LIN {X 0,Y 157.357,Z 221.695,A -85,B 0,C 180,E1 -23600.932,E2 -23600.932} C_VEL
LIN {X 0,Y 157.308,Z 221.703,A -85,B 0,C 180,E1 -23606.678,E2 -23606.678} C_VEL
LIN {X 0,Y 157.277,Z 221.702,A -85,B 0,C 180,E1 -23612.424,E2 -23612.424} C_VEL
LIN {X 0,Y 157.281,Z 221.706,A -85,B 0,C 180,E1 -23616.454,E2 -23616.454} C_VEL
LIN {X 0,Y 157.21,Z 221.714,A -85,B 0,C 180,E1 -23622.107,E2 -23622.107} C_VEL
LIN {X 0,Y 157.207,Z 221.711,A -85,B 0,C 180,E1 -23627.887,E2 -23627.887} C_VEL
LIN {X 0,Y 157.263,Z 221.709,A -85,B 0,C 180,E1 -23633.549,E2 -23633.549} C_VEL
LIN {X 0,Y 157.289,Z 221.703,A -85,B 0,C 180,E1 -23638.094,E2 -23638.094} C_VEL
LIN {X 0,Y 157.317,Z 221.699,A -85,B 0,C 180,E1 -23643.465,E2 -23643.465} C_VEL
LIN {X 0,Y 157.388,Z 221.692,A -85,B 0,C 180,E1 -23649.666,E2 -23649.666} C_VEL
LIN {X 0,Y 157.456,Z 221.679,A -85,B 0,C 180,E1 -23654.466,E2 -23654.466} C_VEL
LIN {X 0,Y 157.728,Z 221.648,A -85,B 0,C 180,E1 -23659.733,E2 -23659.733} C_VEL
LIN {X 0,Y 157.802,Z 221.635,A -85,B 0,C 180,E1 -23662.321,E2 -23662.321} C_VEL
LIN {X 0,Y 158.251,Z 221.58,A -85,B 0,C 180,E1 -23670,E2 -23670} C_VEL
LIN {X 0,Y 157.71,Z 221.652,A -85,B 0,C 180,E1 -23675.113,E2 -23675.113} C_VEL
LIN {X 0,Y 157.744,Z 221.644,A -85,B 0,C 180,E1 -23677.681,E2 -23677.681} C_VEL
LIN {X 0,Y 157.517,Z 221.675,A -85,B 0,C 180,E1 -23681.027,E2 -23681.027} C_VEL
LIN {X 0,Y 156.597,Z 221.813,A -85,B 0,C 180,E1 -23686.708,E2 -23686.708} C_VEL
LIN {X 0,Y 156.129,Z 224.06,A -85,B 0,C 180,E1 -23690.029,E2 -23690.029} C_VEL
LIN {X 0,Y 157.923,Z 235.315,A -85,B 0,C 180,E1 -23691.539,E2 -23691.539} C_VEL
LIN {X 0,Y 159.098,Z 244.23,A -85,B 0,C 180,E1 -23693.081,E2 -23693.081} C_VEL
LIN {X 0,Y 160.081,Z 253.236,A -85,B 0,C 180,E1 -23694.996,E2 -23694.996} C_VEL
LIN {X 0,Y 160.318,Z 256.028,A -85,B 0,C 180,E1 -23695.651,E2 -23695.651} C_VEL
LIN {X 0,Y 159.013,Z 264.361,A -85,B 0,C 180,E1 -23697.883,E2 -23697.883} C_VEL
LIN {X 0,Y 157.724,Z 272.061,A -85,B 0,C 180,E1 -23700.454,E2 -23700.454} C_VEL
LIN {X 0,Y 156.614,Z 279.016,A -85,B 0,C 180,E1 -23703.347,E2 -23703.347} C_VEL
LIN {X 0,Y 155.581,Z 285.499,A -85,B 0,C 180,E1 -23706.765,E2 -23706.765} C_VEL
LIN {X 0,Y 154.989,Z 289.667,A -85,B 0,C 180,E1 -23709.572,E2 -23709.572} C_VEL
LIN {X 0,Y 154.605,Z 293.901,A -85,B 0,C 180,E1 -23713.341,E2 -23713.341} C_VEL
LIN {X 0,Y 154.717,Z 296.859,A -85,B 0,C 180,E1 -23717.053,E2 -23717.053} C_VEL
LIN {X 0,Y 155.31,Z 298.71,A -85,B 0,C 180,E1 -23720.693,E2 -23720.693} C_VEL
LIN {X 0,Y 156.458,Z 299.555,A -85,B 0,C 180,E1 -23724.274,E2 -23724.274} C_VEL
LIN {X 0,Y 158.08,Z 299.423,A -85,B 0,C 180,E1 -23727.761,E2 -23727.761} C_VEL
LIN {X 0,Y 160.289,Z 298.258,A -85,B 0,C 180,E1 -23731.272,E2 -23731.272} C_VEL
LIN {X 0,Y 163.108,Z 295.89,A -85,B 0,C 180,E1 -23734.802,E2 -23734.802} C_VEL
LIN {X 0,Y 166.573,Z 292.371,A -85,B 0,C 180,E1 -23738.158,E2 -23738.158} C_VEL
LIN {X 0,Y 169.515,Z 288.835,A -85,B 0,C 180,E1 -23740.632,E2 -23740.632} C_VEL
LIN {X 0,Y 172.744,Z 284.45,A -85,B 0,C 180,E1 -23743.01,E2 -23743.01} C_VEL
LIN {X 0,Y 175.017,Z 281.08,A -85,B 0,C 180,E1 -23744.523,E2 -23744.523} C_VEL
LIN {X 0,Y 176.013,Z 277.817,A -85,B 0,C 180,E1 -23746.141,E2 -23746.141} C_VEL
LIN {X 0,Y 176.892,Z 271.671,A -85,B 0,C 180,E1 -23749.124,E2 -23749.124} C_VEL
LIN {X 0,Y 176.984,Z 265.582,A -85,B 0,C 180,E1 -23752.013,E2 -23752.013} C_VEL
LIN {X 0,Y 176.219,Z 259.844,A -85,B 0,C 180,E1 -23754.854,E2 -23754.854} C_VEL
LIN {X 0,Y 174.297,Z 253.46,A -85,B 0,C 180,E1 -23758.584,E2 -23758.584} C_VEL
LIN {X 0,Y 172.739,Z 249.567,A -85,B 0,C 180,E1 -23761.168,E2 -23761.168} C_VEL
LIN {X 0,Y 171.244,Z 246.223,A -85,B 0,C 180,E1 -23763.734,E2 -23763.734} C_VEL
LIN {X 0,Y 168.915,Z 243.311,A -85,B 0,C 180,E1 -23767.172,E2 -23767.172} C_VEL
LIN {X 0,Y 167.788,Z 240.918,A -85,B 0,C 180,E1 -23769.647,E2 -23769.647} C_VEL
LIN {X 0,Y 164.941,Z 238.279,A -85,B 0,C 180,E1 -23777.355,E2 -23777.355} C_VEL
LIN {X 0,Y 164.603,Z 237.817,A -85,B 0,C 180,E1 -23780.062,E2 -23780.062} C_VEL
LIN {X 0,Y 164.625,Z 238.233,A -85,B 0,C 180,E1 -23783.929,E2 -23783.929} C_VEL
LIN {X 0,Y 164.925,Z 239.123,A -85,B 0,C 180,E1 -23786.508,E2 -23786.508} C_VEL
LIN {X 0,Y 167.958,Z 244.088,A -85,B 0,C 180,E1 -23794.624,E2 -23794.624} C_VEL
LIN {X 0,Y 169.814,Z 248.809,A -85,B 0,C 180,E1 -23798.376,E2 -23798.376} C_VEL
LIN {X 0,Y 170.797,Z 250.242,A -85,B 0,C 180,E1 -23799.699,E2 -23799.699} C_VEL
LIN {X 0,Y 173.191,Z 256.311,A -85,B 0,C 180,E1 -23803.621,E2 -23803.621} C_VEL
LIN {X 0,Y 175.702,Z 263.842,A -85,B 0,C 180,E1 -23807.731,E2 -23807.731} C_VEL
LIN {X 0,Y 176.827,Z 268.296,A -85,B 0,C 180,E1 -23809.866,E2 -23809.866} C_VEL
LIN {X 0,Y 176.722,Z 272.386,A -85,B 0,C 180,E1 -23811.419,E2 -23811.419} C_VEL
LIN {X 0,Y 175.572,Z 280.289,A -85,B 0,C 180,E1 -23814.316,E2 -23814.316} C_VEL
LIN {X 0,Y 173.444,Z 288.286,A -85,B 0,C 180,E1 -23817.528,E2 -23817.528} C_VEL
LIN {X 0,Y 171.758,Z 292.829,A -85,B 0,C 180,E1 -23819.555,E2 -23819.555} C_VEL
LIN {X 0,Y 168.933,Z 297.944,A -85,B 0,C 180,E1 -23822.094,E2 -23822.094} C_VEL
LIN {X 0,Y 165.345,Z 302.617,A -85,B 0,C 180,E1 -23824.846,E2 -23824.846} C_VEL
LIN {X 0,Y 161.783,Z 306.868,A -85,B 0,C 180,E1 -23828.331,E2 -23828.331} C_VEL
LIN {X 0,Y 158.947,Z 309.905,A -85,B 0,C 180,E1 -23831.971,E2 -23831.971} C_VEL
LIN {X 0,Y 157.539,Z 311.3,A -85,B 0,C 180,E1 -23834.475,E2 -23834.475} C_VEL
LIN {X 0,Y 156.396,Z 312.246,A -85,B 0,C 180,E1 -23837.016,E2 -23837.016} C_VEL
LIN {X 0,Y 155.614,Z 312.675,A -85,B 0,C 180,E1 -23839.593,E2 -23839.593} C_VEL
LIN {X 0,Y 155.132,Z 312.568,A -85,B 0,C 180,E1 -23842.189,E2 -23842.189} C_VEL
LIN {X 0,Y 154.948,Z 311.55,A -85,B 0,C 180,E1 -23846.274,E2 -23846.274} C_VEL
LIN {X 0,Y 155.245,Z 309.496,A -85,B 0,C 180,E1 -23850,E2 -23850} C_VEL
LIN {X 0,Y 155.182,Z 306.489,A -85,B 0,C 180,E1 -23853.423,E2 -23853.423} C_VEL
LIN {X 0,Y 155.219,Z 302.834,A -85,B 0,C 180,E1 -23856.5,E2 -23856.5} C_VEL
LIN {X 0,Y 155.653,Z 297.85,A -85,B 0,C 180,E1 -23859.749,E2 -23859.749} C_VEL
LIN {X 0,Y 156.199,Z 292.931,A -85,B 0,C 180,E1 -23862.341,E2 -23862.341} C_VEL
LIN {X 0,Y 157.058,Z 286.99,A -85,B 0,C 180,E1 -23864.91,E2 -23864.91} C_VEL
LIN {X 0,Y 158.18,Z 279.751,A -85,B 0,C 180,E1 -23867.452,E2 -23867.452} C_VEL
LIN {X 0,Y 158.643,Z 275.533,A -85,B 0,C 180,E1 -23868.735,E2 -23868.735} C_VEL
LIN {X 0,Y 158.451,Z 266.744,A -85,B 0,C 180,E1 -23870.973,E2 -23870.973} C_VEL
LIN {X 0,Y 158.166,Z 258.965,A -85,B 0,C 180,E1 -23872.606,E2 -23872.606} C_VEL
LIN {X 0,Y 157.761,Z 249.777,A -85,B 0,C 180,E1 -23874.161,E2 -23874.161} C_VEL
LIN {X 0,Y 157.069,Z 239.045,A -85,B 0,C 180,E1 -23875.555,E2 -23875.555} C_VEL
LIN {X 0,Y 156.809,Z 235.295,A -85,B 0,C 180,E1 -23875.97,E2 -23875.97} C_VEL
LIN {X 0,Y 158.126,Z 231.22,A -85,B 0,C 180,E1 -23880.739,E2 -23880.739} C_VEL
LIN {X 0,Y 158.843,Z 228.659,A -85,B 0,C 180,E1 -23883.759,E2 -23883.759} C_VEL
LIN {X 0,Y 157.955,Z 224.322,A -85,B 0,C 180,E1 -23889.248,E2 -23889.248} C_VEL
LIN {X 0,Y 156.982,Z 223.117,A -85,B 0,C 180,E1 -23891.311,E2 -23891.311} C_VEL
LIN {X 0,Y 155.184,Z 222.534,A -85,B 0,C 180,E1 -23893.376,E2 -23893.376} C_VEL
LIN {X 0,Y 151.248,Z 222.465,A -85,B 0,C 180,E1 -23897.633,E2 -23897.633} C_VEL
LIN {X 0,Y 150.18,Z 222.59,A -85,B 0,C 180,E1 -23899.886,E2 -23899.886} C_VEL
LIN {X 0,Y 150.096,Z 222.591,A -85,B 0,C 180,E1 -23900.651,E2 -23900.651} C_VEL
LIN {X 0,Y 150.194,Z 222.584,A -85,B 0,C 180,E1 -23905.837,E2 -23905.837} C_VEL
LIN {X 0,Y 150.21,Z 222.586,A -85,B 0,C 180,E1 -23909.023,E2 -23909.023} C_VEL
LIN {X 0,Y 150.246,Z 222.576,A -85,B 0,C 180,E1 -23912.719,E2 -23912.719} C_VEL
LIN {X 0,Y 150.354,Z 222.568,A -85,B 0,C 180,E1 -23919.207,E2 -23919.207} C_VEL
LIN {X 0,Y 150.366,Z 222.566,A -85,B 0,C 180,E1 -23923.712,E2 -23923.712} C_VEL
LIN {X 0,Y 150.615,Z 222.532,A -85,B 0,C 180,E1 -23929.241,E2 -23929.241} C_VEL
LIN {X 0,Y 150.707,Z 222.523,A -85,B 0,C 180,E1 -23931.956,E2 -23931.956} C_VEL
LIN {X 0,Y 151.22,Z 222.458,A -85,B 0,C 180,E1 -23939.998,E2 -23939.998} C_VEL
LIN {X 0,Y 150.706,Z 222.521,A -85,B 0,C 180,E1 -23948.04,E2 -23948.04} C_VEL
LIN {X 0,Y 150.576,Z 222.54,A -85,B 0,C 180,E1 -23951.43,E2 -23951.43} C_VEL
LIN {X 0,Y 150.329,Z 222.568,A -85,B 0,C 180,E1 -23956.288,E2 -23956.288} C_VEL
LIN {X 0,Y 150.339,Z 222.57,A -85,B 0,C 180,E1 -23960.777,E2 -23960.777} C_VEL
LIN {X 0,Y 150.24,Z 222.582,A -85,B 0,C 180,E1 -23967.277,E2 -23967.277} C_VEL
LIN {X 0,Y 150.217,Z 222.583,A -85,B 0,C 180,E1 -23972.632,E2 -23972.632} C_VEL
LIN {X 0,Y 150.209,Z 222.586,A -85,B 0,C 180,E1 -23977.459,E2 -23977.459} C_VEL
LIN {X 0,Y 150.151,Z 222.59,A -85,B 0,C 180,E1 -23981.504,E2 -23981.504} C_VEL
LIN {X 0,Y 150.122,Z 222.597,A -85,B 0,C 180,E1 -23985.393,E2 -23985.393} C_VEL
LIN {X 0,Y 150.146,Z 222.589,A -85,B 0,C 180,E1 -23989.056,E2 -23989.056} C_VEL
LIN {X 0,Y 150.175,Z 222.59,A -85,B 0,C 180,E1 -23992.705,E2 -23992.705} C_VEL
LIN {X 0,Y 150.21,Z 222.581,A -85,B 0,C 180,E1 -23997.366,E2 -23997.366} C_VEL
LIN {X 0,Y 150.239,Z 222.581,A -85,B 0,C 180,E1 -24002.716,E2 -24002.716} C_VEL
LIN {X 0,Y 150.345,Z 222.571,A -85,B 0,C 180,E1 -24009.206,E2 -24009.206} C_VEL
LIN {X 0,Y 150.362,Z 222.563,A -85,B 0,C 180,E1 -24013.713,E2 -24013.713} C_VEL
LIN {X 0,Y 150.652,Z 222.53,A -85,B 0,C 180,E1 -24019.245,E2 -24019.245} C_VEL
LIN {X 0,Y 150.738,Z 222.514,A -85,B 0,C 180,E1 -24021.959,E2 -24021.959} C_VEL
LIN {X 0,Y 151.211,Z 222.456,A -85,B 0,C 180,E1 -24030,E2 -24030} C_VEL
LIN {X 0,Y 150.654,Z 222.527,A -85,B 0,C 180,E1 -24038.044,E2 -24038.044} C_VEL
LIN {X 0,Y 150.433,Z 222.558,A -85,B 0,C 180,E1 -24041.177,E2 -24041.177} C_VEL
LIN {X 0,Y 149.471,Z 222.712,A -85,B 0,C 180,E1 -24046.913,E2 -24046.913} C_VEL
LIN {X 0,Y 149.11,Z 224.303,A -85,B 0,C 180,E1 -24049.354,E2 -24049.354} C_VEL
LIN {X 0,Y 150.794,Z 234.895,A -85,B 0,C 180,E1 -24050.816,E2 -24050.816} C_VEL
LIN {X 0,Y 151.854,Z 242.993,A -85,B 0,C 180,E1 -24052.245,E2 -24052.245} C_VEL
LIN {X 0,Y 152.818,Z 251.392,A -85,B 0,C 180,E1 -24054.053,E2 -24054.053} C_VEL
LIN {X 0,Y 153.211,Z 257.128,A -85,B 0,C 180,E1 -24055.47,E2 -24055.47} C_VEL
LIN {X 0,Y 151.953,Z 264.547,A -85,B 0,C 180,E1 -24057.549,E2 -24057.549} C_VEL
LIN {X 0,Y 150.658,Z 272.211,A -85,B 0,C 180,E1 -24060.216,E2 -24060.216} C_VEL
LIN {X 0,Y 149.479,Z 279.357,A -85,B 0,C 180,E1 -24063.322,E2 -24063.322} C_VEL
LIN {X 0,Y 148.373,Z 286.201,A -85,B 0,C 180,E1 -24067.166,E2 -24067.166} C_VEL
LIN {X 0,Y 147.739,Z 290.657,A -85,B 0,C 180,E1 -24070.441,E2 -24070.441} C_VEL
LIN {X 0,Y 147.492,Z 294.709,A -85,B 0,C 180,E1 -24074.381,E2 -24074.381} C_VEL
LIN {X 0,Y 147.734,Z 297.522,A -85,B 0,C 180,E1 -24078.244,E2 -24078.244} C_VEL
LIN {X 0,Y 148.531,Z 299.257,A -85,B 0,C 180,E1 -24082.043,E2 -24082.043} C_VEL
LIN {X 0,Y 149.895,Z 299.978,A -85,B 0,C 180,E1 -24085.765,E2 -24085.765} C_VEL
LIN {X 0,Y 151.779,Z 299.699,A -85,B 0,C 180,E1 -24089.383,E2 -24089.383} C_VEL
LIN {X 0,Y 154.19,Z 298.452,A -85,B 0,C 180,E1 -24092.886,E2 -24092.886} C_VEL
LIN {X 0,Y 157.064,Z 296.25,A -85,B 0,C 180,E1 -24096.255,E2 -24096.255} C_VEL
LIN {X 0,Y 160.567,Z 292.975,A -85,B 0,C 180,E1 -24099.505,E2 -24099.505} C_VEL
LIN {X 0,Y 164.43,Z 288.619,A -85,B 0,C 180,E1 -24102.593,E2 -24102.593} C_VEL
LIN {X 0,Y 168.84,Z 282.94,A -85,B 0,C 180,E1 -24105.539,E2 -24105.539} C_VEL
LIN {X 0,Y 170.062,Z 279.332,A -85,B 0,C 180,E1 -24107.472,E2 -24107.472} C_VEL
LIN {X 0,Y 171.082,Z 273.883,A -85,B 0,C 180,E1 -24110.37,E2 -24110.37} C_VEL
LIN {X 0,Y 171.363,Z 268.962,A -85,B 0,C 180,E1 -24112.935,E2 -24112.935} C_VEL
LIN {X 0,Y 171.142,Z 264.718,A -85,B 0,C 180,E1 -24115.291,E2 -24115.291} C_VEL
LIN {X 0,Y 169.882,Z 259.168,A -85,B 0,C 180,E1 -24118.817,E2 -24118.817} C_VEL
LIN {X 0,Y 168.254,Z 254.292,A -85,B 0,C 180,E1 -24122.396,E2 -24122.396} C_VEL
LIN {X 0,Y 167.637,Z 252.581,A -85,B 0,C 180,E1 -24123.814,E2 -24123.814} C_VEL
LIN {X 0,Y 164.769,Z 247.382,A -85,B 0,C 180,E1 -24129.826,E2 -24129.826} C_VEL
LIN {X 0,Y 162.267,Z 244.828,A -85,B 0,C 180,E1 -24137.665,E2 -24137.665} C_VEL
LIN {X 0,Y 162.024,Z 244.453,A -85,B 0,C 180,E1 -24140.307,E2 -24140.307} C_VEL
LIN {X 0,Y 162.115,Z 245.007,A -85,B 0,C 180,E1 -24144.441,E2 -24144.441} C_VEL
LIN {X 0,Y 162.645,Z 246.843,A -85,B 0,C 180,E1 -24148.382,E2 -24148.382} C_VEL
LIN {X 0,Y 164.582,Z 250.059,A -85,B 0,C 180,E1 -24153.722,E2 -24153.722} C_VEL
LIN {X 0,Y 166.942,Z 256.043,A -85,B 0,C 180,E1 -24159.161,E2 -24159.161} C_VEL
LIN {X 0,Y 168.757,Z 261.525,A -85,B 0,C 180,E1 -24162.984,E2 -24162.984} C_VEL
LIN {X 0,Y 170.316,Z 267.016,A -85,B 0,C 180,E1 -24166.231,E2 -24166.231} C_VEL
LIN {X 0,Y 171.4,Z 272.056,A -85,B 0,C 180,E1 -24169.001,E2 -24169.001} C_VEL
LIN {X 0,Y 171.045,Z 275.831,A -85,B 0,C 180,E1 -24170.555,E2 -24170.555} C_VEL
LIN {X 0,Y 169.552,Z 282.828,A -85,B 0,C 180,E1 -24173.393,E2 -24173.393} C_VEL
LIN {X 0,Y 167.996,Z 287.976,A -85,B 0,C 180,E1 -24175.615,E2 -24175.615} C_VEL
LIN {X 0,Y 165.588,Z 293.793,A -85,B 0,C 180,E1 -24178.393,E2 -24178.393} C_VEL
LIN {X 0,Y 163.418,Z 297.577,A -85,B 0,C 180,E1 -24180.359,E2 -24180.359} C_VEL
LIN {X 0,Y 158.967,Z 302.982,A -85,B 0,C 180,E1 -24183.762,E2 -24183.762} C_VEL
LIN {X 0,Y 155.217,Z 307.043,A -85,B 0,C 180,E1 -24187.365,E2 -24187.365} C_VEL
LIN {X 0,Y 152.191,Z 309.927,A -85,B 0,C 180,E1 -24191.141,E2 -24191.141} C_VEL
LIN {X 0,Y 150.691,Z 311.177,A -85,B 0,C 180,E1 -24193.75,E2 -24193.75} C_VEL
LIN {X 0,Y 149.48,Z 311.981,A -85,B 0,C 180,E1 -24196.404,E2 -24196.404} C_VEL
LIN {X 0,Y 148.616,Z 312.347,A -85,B 0,C 180,E1 -24199.097,E2 -24199.097} C_VEL
LIN {X 0,Y 148.085,Z 312.163,A -85,B 0,C 180,E1 -24201.815,E2 -24201.815} C_VEL
LIN {X 0,Y 147.889,Z 310.828,A -85,B 0,C 180,E1 -24206.368,E2 -24206.368} C_VEL
LIN {X 0,Y 148.186,Z 308.713,A -85,B 0,C 180,E1 -24210.001,E2 -24210.001} C_VEL
LIN {X 0,Y 148.14,Z 305.73,A -85,B 0,C 180,E1 -24213.412,E2 -24213.412} C_VEL
LIN {X 0,Y 148.183,Z 301.724,A -85,B 0,C 180,E1 -24216.81,E2 -24216.81} C_VEL
LIN {X 0,Y 148.656,Z 296.56,A -85,B 0,C 180,E1 -24220.212,E2 -24220.212} C_VEL
LIN {X 0,Y 149.262,Z 291.444,A -85,B 0,C 180,E1 -24222.924,E2 -24222.924} C_VEL
LIN {X 0,Y 150.193,Z 285.274,A -85,B 0,C 180,E1 -24225.609,E2 -24225.609} C_VEL
LIN {X 0,Y 151.502,Z 276.74,A -85,B 0,C 180,E1 -24228.598,E2 -24228.598} C_VEL
LIN {X 0,Y 151.432,Z 267.772,A -85,B 0,C 180,E1 -24231.081,E2 -24231.081} C_VEL
LIN {X 0,Y 151.15,Z 259.634,A -85,B 0,C 180,E1 -24232.918,E2 -24232.918} C_VEL
LIN {X 0,Y 150.775,Z 250.215,A -85,B 0,C 180,E1 -24234.621,E2 -24234.621} C_VEL
LIN {X 0,Y 150.204,Z 240.494,A -85,B 0,C 180,E1 -24235.984,E2 -24235.984} C_VEL
LIN {X 0,Y 149.858,Z 235.041,A -85,B 0,C 180,E1 -24236.662,E2 -24236.662} C_VEL
LIN {X 0,Y 151.413,Z 230.571,A -85,B 0,C 180,E1 -24242.123,E2 -24242.123} C_VEL
LIN {X 0,Y 151.753,Z 229.253,A -85,B 0,C 180,E1 -24243.763,E2 -24243.763} C_VEL
LIN {X 0,Y 151.135,Z 226.209,A -85,B 0,C 180,E1 -24247.763,E2 -24247.763} C_VEL
LIN {X 0,Y 150.464,Z 222.555,A -85,B 0,C 180,E1 -24252.807,E2 -24252.807} C_VEL
LIN {X 0,Y 150.154,Z 222.592,A -85,B 0,C 180,E1 -24259.057,E2 -24259.057} C_VEL
LIN {X 0,Y 150.096,Z 222.591,A -85,B 0,C 180,E1 -24260.651,E2 -24260.651} C_VEL
LIN {X 0,Y 149.455,Z 222.68,A -85,B 0,C 180,E1 -24262.891,E2 -24262.891} C_VEL
LIN {X 0,Y 147.93,Z 222.869,A -85,B 0,C 180,E1 -24265.102,E2 -24265.102} C_VEL
LIN {X 0,Y 143.499,Z 223.421,A -85,B 0,C 180,E1 -24271.171,E2 -24271.171} C_VEL
LIN {X 0,Y 143.163,Z 223.458,A -85,B 0,C 180,E1 -24272.77,E2 -24272.77} C_VEL
LIN {X 0,Y 143.28,Z 223.448,A -85,B 0,C 180,E1 -24278.746,E2 -24278.746} C_VEL
LIN {X 0,Y 143.305,Z 223.442,A -85,B 0,C 180,E1 -24282.885,E2 -24282.885} C_VEL
LIN {X 0,Y 143.541,Z 223.414,A -85,B 0,C 180,E1 -24288.703,E2 -24288.703} C_VEL
LIN {X 0,Y 143.629,Z 223.404,A -85,B 0,C 180,E1 -24291.556,E2 -24291.556} C_VEL
LIN {X 0,Y 144.178,Z 223.335,A -85,B 0,C 180,E1 -24299.998,E2 -24299.998} C_VEL
LIN {X 0,Y 143.627,Z 223.403,A -85,B 0,C 180,E1 -24308.439,E2 -24308.439} C_VEL
LIN {X 0,Y 143.502,Z 223.421,A -85,B 0,C 180,E1 -24311.618,E2 -24311.618} C_VEL
LIN {X 0,Y 143.268,Z 223.451,A -85,B 0,C 180,E1 -24317.115,E2 -24317.115} C_VEL
LIN {X 0,Y 143.267,Z 223.449,A -85,B 0,C 180,E1 -24321.242,E2 -24321.242} C_VEL
LIN {X 0,Y 143.187,Z 223.461,A -85,B 0,C 180,E1 -24327.933,E2 -24327.933} C_VEL
LIN {X 0,Y 143.167,Z 223.461,A -85,B 0,C 180,E1 -24333.433,E2 -24333.433} C_VEL
LIN {X 0,Y 143.072,Z 223.471,A -85,B 0,C 180,E1 -24339.683,E2 -24339.683} C_VEL
LIN {X 0,Y 143.054,Z 223.477,A -85,B 0,C 180,E1 -24343.452,E2 -24343.452} C_VEL
LIN {X 0,Y 143.061,Z 223.474,A -85,B 0,C 180,E1 -24347.463,E2 -24347.463} C_VEL
LIN {X 0,Y 143.073,Z 223.476,A -85,B 0,C 180,E1 -24351.804,E2 -24351.804} C_VEL
LIN {X 0,Y 143.177,Z 223.457,A -85,B 0,C 180,E1 -24357.319,E2 -24357.319} C_VEL
LIN {X 0,Y 143.186,Z 223.46,A -85,B 0,C 180,E1 -24362.061,E2 -24362.061} C_VEL
LIN {X 0,Y 143.271,Z 223.45,A -85,B 0,C 180,E1 -24368.744,E2 -24368.744} C_VEL
LIN {X 0,Y 143.299,Z 223.443,A -85,B 0,C 180,E1 -24372.886,E2 -24372.886} C_VEL
LIN {X 0,Y 143.588,Z 223.412,A -85,B 0,C 180,E1 -24378.709,E2 -24378.709} C_VEL
LIN {X 0,Y 143.659,Z 223.396,A -85,B 0,C 180,E1 -24381.56,E2 -24381.56} C_VEL
LIN {X 0,Y 144.17,Z 223.333,A -85,B 0,C 180,E1 -24389.999,E2 -24389.999} C_VEL
LIN {X 0,Y 143.565,Z 223.409,A -85,B 0,C 180,E1 -24398.445,E2 -24398.445} C_VEL
LIN {X 0,Y 143.336,Z 223.441,A -85,B 0,C 180,E1 -24401.31,E2 -24401.31} C_VEL
LIN {X 0,Y 142.382,Z 223.56,A -85,B 0,C 180,E1 -24407.042,E2 -24407.042} C_VEL
LIN {X 0,Y 142.126,Z 224.534,A -85,B 0,C 180,E1 -24408.628,E2 -24408.628} C_VEL
LIN {X 0,Y 143.95,Z 236.408,A -85,B 0,C 180,E1 -24410.421,E2 -24410.421} C_VEL
LIN {X 0,Y 145.022,Z 244.991,A -85,B 0,C 180,E1 -24412.06,E2 -24412.06} C_VEL
LIN {X 0,Y 145.95,Z 253.361,A -85,B 0,C 180,E1 -24414.01,E2 -24414.01} C_VEL
LIN {X 0,Y 146.104,Z 257.993,A -85,B 0,C 180,E1 -24415.233,E2 -24415.233} C_VEL
LIN {X 0,Y 144.766,Z 265.459,A -85,B 0,C 180,E1 -24417.464,E2 -24417.464} C_VEL
LIN {X 0,Y 143.528,Z 272.666,A -85,B 0,C 180,E1 -24420.125,E2 -24420.125} C_VEL
LIN {X 0,Y 142.175,Z 280.577,A -85,B 0,C 180,E1 -24423.785,E2 -24423.785} C_VEL
LIN {X 0,Y 141.092,Z 287.245,A -85,B 0,C 180,E1 -24427.903,E2 -24427.903} C_VEL
LIN {X 0,Y 140.525,Z 291.614,A -85,B 0,C 180,E1 -24431.398,E2 -24431.398} C_VEL
LIN {X 0,Y 140.414,Z 295.51,A -85,B 0,C 180,E1 -24435.519,E2 -24435.519} C_VEL
LIN {X 0,Y 140.823,Z 298.186,A -85,B 0,C 180,E1 -24439.554,E2 -24439.554} C_VEL
LIN {X 0,Y 141.844,Z 299.78,A -85,B 0,C 180,E1 -24443.521,E2 -24443.521} C_VEL
LIN {X 0,Y 143.445,Z 300.35,A -85,B 0,C 180,E1 -24447.392,E2 -24447.392} C_VEL
LIN {X 0,Y 145.616,Z 299.941,A -85,B 0,C 180,E1 -24451.145,E2 -24451.145} C_VEL
LIN {X 0,Y 148.329,Z 298.586,A -85,B 0,C 180,E1 -24454.762,E2 -24454.762} C_VEL
LIN {X 0,Y 151.549,Z 296.269,A -85,B 0,C 180,E1 -24458.226,E2 -24458.226} C_VEL
LIN {X 0,Y 155.317,Z 292.905,A -85,B 0,C 180,E1 -24461.536,E2 -24461.536} C_VEL
LIN {X 0,Y 160.083,Z 287.925,A -85,B 0,C 180,E1 -24464.982,E2 -24464.982} C_VEL
LIN {X 0,Y 163.095,Z 284.085,A -85,B 0,C 180,E1 -24466.988,E2 -24466.988} C_VEL
LIN {X 0,Y 164.871,Z 278.73,A -85,B 0,C 180,E1 -24470.185,E2 -24470.185} C_VEL
LIN {X 0,Y 165.739,Z 273.335,A -85,B 0,C 180,E1 -24473.306,E2 -24473.306} C_VEL
LIN {X 0,Y 165.75,Z 268.349,A -85,B 0,C 180,E1 -24476.356,E2 -24476.356} C_VEL
LIN {X 0,Y 164.829,Z 263.239,A -85,B 0,C 180,E1 -24480.002,E2 -24480.002} C_VEL
LIN {X 0,Y 163.638,Z 258.825,A -85,B 0,C 180,E1 -24483.696,E2 -24483.696} C_VEL
LIN {X 0,Y 162.566,Z 256.708,A -85,B 0,C 180,E1 -24486.109,E2 -24486.109} C_VEL
LIN {X 0,Y 161.318,Z 253.617,A -85,B 0,C 180,E1 -24490.038,E2 -24490.038} C_VEL
LIN {X 0,Y 159.191,Z 251.178,A -85,B 0,C 180,E1 -24498.003,E2 -24498.003} C_VEL
LIN {X 0,Y 159.005,Z 251.007,A -85,B 0,C 180,E1 -24501.846,E2 -24501.846} C_VEL
LIN {X 0,Y 159.075,Z 251.221,A -85,B 0,C 180,E1 -24503.432,E2 -24503.432} C_VEL
LIN {X 0,Y 159.204,Z 252.152,A -85,B 0,C 180,E1 -24506.198,E2 -24506.198} C_VEL
LIN {X 0,Y 160.382,Z 255.147,A -85,B 0,C 180,E1 -24511.727,E2 -24511.727} C_VEL
LIN {X 0,Y 161.35,Z 257.328,A -85,B 0,C 180,E1 -24514.491,E2 -24514.491} C_VEL
LIN {X 0,Y 162.876,Z 262.191,A -85,B 0,C 180,E1 -24519.042,E2 -24519.042} C_VEL
LIN {X 0,Y 164.073,Z 266.36,A -85,B 0,C 180,E1 -24522.182,E2 -24522.182} C_VEL
LIN {X 0,Y 165.431,Z 272.608,A -85,B 0,C 180,E1 -24526.24,E2 -24526.24} C_VEL
LIN {X 0,Y 165.855,Z 275.249,A -85,B 0,C 180,E1 -24527.879,E2 -24527.879} C_VEL
LIN {X 0,Y 165.269,Z 279.337,A -85,B 0,C 180,E1 -24529.733,E2 -24529.733} C_VEL
LIN {X 0,Y 163.201,Z 286.494,A -85,B 0,C 180,E1 -24532.923,E2 -24532.923} C_VEL
LIN {X 0,Y 160.103,Z 293.616,A -85,B 0,C 180,E1 -24536.519,E2 -24536.519} C_VEL
LIN {X 0,Y 157.306,Z 298.17,A -85,B 0,C 180,E1 -24539.084,E2 -24539.084} C_VEL
LIN {X 0,Y 152.654,Z 303.37,A -85,B 0,C 180,E1 -24542.588,E2 -24542.588} C_VEL
LIN {X 0,Y 148.701,Z 307.261,A -85,B 0,C 180,E1 -24546.314,E2 -24546.314} C_VEL
LIN {X 0,Y 145.473,Z 309.961,A -85,B 0,C 180,E1 -24550.234,E2 -24550.234} C_VEL
LIN {X 0,Y 143.876,Z 311.06,A -85,B 0,C 180,E1 -24552.958,E2 -24552.958} C_VEL
LIN {X 0,Y 142.589,Z 311.717,A -85,B 0,C 180,E1 -24555.733,E2 -24555.733} C_VEL
LIN {X 0,Y 141.642,Z 311.944,A -85,B 0,C 180,E1 -24558.553,E2 -24558.553} C_VEL
LIN {X 0,Y 141.048,Z 311.72,A -85,B 0,C 180,E1 -24561.404,E2 -24561.404} C_VEL
LIN {X 0,Y 140.85,Z 310.051,A -85,B 0,C 180,E1 -24566.351,E2 -24566.351} C_VEL
LIN {X 0,Y 141.127,Z 307.88,A -85,B 0,C 180,E1 -24570.001,E2 -24570.001} C_VEL
LIN {X 0,Y 141.121,Z 305.505,A -85,B 0,C 180,E1 -24572.855,E2 -24572.855} C_VEL
LIN {X 0,Y 141.054,Z 302.461,A -85,B 0,C 180,E1 -24575.72,E2 -24575.72} C_VEL
LIN {X 0,Y 141.426,Z 297.571,A -85,B 0,C 180,E1 -24579.295,E2 -24579.295} C_VEL
LIN {X 0,Y 141.979,Z 292.756,A -85,B 0,C 180,E1 -24582.145,E2 -24582.145} C_VEL
LIN {X 0,Y 142.812,Z 286.904,A -85,B 0,C 180,E1 -24584.973,E2 -24584.973} C_VEL
LIN {X 0,Y 143.987,Z 279.782,A -85,B 0,C 180,E1 -24587.762,E2 -24587.762} C_VEL
LIN {X 0,Y 144.464,Z 275.668,A -85,B 0,C 180,E1 -24589.171,E2 -24589.171} C_VEL
LIN {X 0,Y 144.326,Z 266.004,A -85,B 0,C 180,E1 -24591.89,E2 -24591.89} C_VEL
LIN {X 0,Y 144.066,Z 257.989,A -85,B 0,C 180,E1 -24593.733,E2 -24593.733} C_VEL
LIN {X 0,Y 143.745,Z 249.405,A -85,B 0,C 180,E1 -24595.329,E2 -24595.329} C_VEL
LIN {X 0,Y 143.193,Z 239.472,A -85,B 0,C 180,E1 -24596.762,E2 -24596.762} C_VEL
LIN {X 0,Y 142.909,Z 234.747,A -85,B 0,C 180,E1 -24597.394,E2 -24597.394} C_VEL
LIN {X 0,Y 144.357,Z 230.89,A -85,B 0,C 180,E1 -24602.381,E2 -24602.381} C_VEL
LIN {X 0,Y 144.6,Z 229.445,A -85,B 0,C 180,E1 -24604.281,E2 -24604.281} C_VEL
LIN {X 0,Y 143.819,Z 225.744,A -85,B 0,C 180,E1 -24609.441,E2 -24609.441} C_VEL
LIN {X 0,Y 143.427,Z 223.431,A -85,B 0,C 180,E1 -24612.884,E2 -24612.884} C_VEL
LIN {X 0,Y 143.065,Z 223.478,A -85,B 0,C 180,E1 -24620.308,E2 -24620.308} C_VEL
LIN {X 0,Y 143.168,Z 223.462,A -85,B 0,C 180,E1 -24626.566,E2 -24626.566} C_VEL
LIN {X 0,Y 143.163,Z 223.458,A -85,B 0,C 180,E1 -24632.77,E2 -24632.77} C_VEL
LIN {X 0,Y 142.472,Z 223.549,A -85,B 0,C 180,E1 -24635.118,E2 -24635.118} C_VEL
LIN {X 0,Y 140.921,Z 223.747,A -85,B 0,C 180,E1 -24637.437,E2 -24637.437} C_VEL
LIN {X 0,Y 136.556,Z 224.292,A -85,B 0,C 180,E1 -24643.817,E2 -24643.817} C_VEL
LIN {X 0,Y 136.273,Z 224.319,A -85,B 0,C 180,E1 -24645.497,E2 -24645.497} C_VEL
LIN {X 0,Y 136.449,Z 224.298,A -85,B 0,C 180,E1 -24648.136,E2 -24648.136} C_VEL
LIN {X 0,Y 136.555,Z 224.283,A -85,B 0,C 180,E1 -24651.116,E2 -24651.116} C_VEL
LIN {X 0,Y 137.135,Z 224.213,A -85,B 0,C 180,E1 -24659.997,E2 -24659.997} C_VEL
LIN {X 0,Y 136.552,Z 224.286,A -85,B 0,C 180,E1 -24668.88,E2 -24668.88} C_VEL
LIN {X 0,Y 136.417,Z 224.304,A -85,B 0,C 180,E1 -24671.89,E2 -24671.89} C_VEL
LIN {X 0,Y 136.188,Z 224.332,A -85,B 0,C 180,E1 -24678.034,E2 -24678.034} C_VEL
LIN {X 0,Y 136.189,Z 224.33,A -85,B 0,C 180,E1 -24681.737,E2 -24681.737} C_VEL
LIN {X 0,Y 136.113,Z 224.342,A -85,B 0,C 180,E1 -24688.624,E2 -24688.624} C_VEL
LIN {X 0,Y 136.077,Z 224.347,A -85,B 0,C 180,E1 -24694.616,E2 -24694.616} C_VEL
LIN {X 0,Y 136.048,Z 224.346,A -85,B 0,C 180,E1 -24699.205,E2 -24699.205} C_VEL
LIN {X 0,Y 135.995,Z 224.357,A -85,B 0,C 180,E1 -24703.655,E2 -24703.655} C_VEL
LIN {X 0,Y 136.001,Z 224.352,A -85,B 0,C 180,E1 -24707.794,E2 -24707.794} C_VEL
LIN {X 0,Y 136.023,Z 224.354,A -85,B 0,C 180,E1 -24711.682,E2 -24711.682} C_VEL
LIN {X 0,Y 136.051,Z 224.346,A -85,B 0,C 180,E1 -24715.737,E2 -24715.737} C_VEL
LIN {X 0,Y 136.142,Z 224.338,A -85,B 0,C 180,E1 -24722.315,E2 -24722.315} C_VEL
LIN {X 0,Y 136.238,Z 224.327,A -85,B 0,C 180,E1 -24728.831,E2 -24728.831} C_VEL
LIN {X 0,Y 136.27,Z 224.32,A -85,B 0,C 180,E1 -24735.056,E2 -24735.056} C_VEL
LIN {X 0,Y 136.491,Z 224.295,A -85,B 0,C 180,E1 -24738.114,E2 -24738.114} C_VEL
LIN {X 0,Y 136.586,Z 224.278,A -85,B 0,C 180,E1 -24741.119,E2 -24741.119} C_VEL
LIN {X 0,Y 137.127,Z 224.21,A -85,B 0,C 180,E1 -24749.999,E2 -24749.999} C_VEL
LIN {X 0,Y 136.528,Z 224.29,A -85,B 0,C 180,E1 -24755.909,E2 -24755.909} C_VEL
LIN {X 0,Y 136.466,Z 224.294,A -85,B 0,C 180,E1 -24758.887,E2 -24758.887} C_VEL
LIN {X 0,Y 136.15,Z 224.337,A -85,B 0,C 180,E1 -24761.915,E2 -24761.915} C_VEL
LIN {X 0,Y 135.311,Z 224.44,A -85,B 0,C 180,E1 -24766.987,E2 -24766.987} C_VEL
LIN {X 0,Y 135.148,Z 224.803,A -85,B 0,C 180,E1 -24767.886,E2 -24767.886} C_VEL
LIN {X 0,Y 136.773,Z 235.484,A -85,B 0,C 180,E1 -24769.532,E2 -24769.532} C_VEL
LIN {X 0,Y 137.936,Z 244.668,A -85,B 0,C 180,E1 -24771.354,E2 -24771.354} C_VEL
LIN {X 0,Y 138.903,Z 253.821,A -85,B 0,C 180,E1 -24773.588,E2 -24773.588} C_VEL
LIN {X 0,Y 139.149,Z 257.583,A -85,B 0,C 180,E1 -24774.622,E2 -24774.622} C_VEL
LIN {X 0,Y 137.581,Z 266.308,A -85,B 0,C 180,E1 -24777.37,E2 -24777.37} C_VEL
LIN {X 0,Y 136.429,Z 272.812,A -85,B 0,C 180,E1 -24779.902,E2 -24779.902} C_VEL
LIN {X 0,Y 135.295,Z 279.364,A -85,B 0,C 180,E1 -24783.027,E2 -24783.027} C_VEL
LIN {X 0,Y 134.283,Z 285.314,A -85,B 0,C 180,E1 -24786.551,E2 -24786.551} C_VEL
LIN {X 0,Y 133.519,Z 290.842,A -85,B 0,C 180,E1 -24790.779,E2 -24790.779} C_VEL
LIN {X 0,Y 133.316,Z 294.892,A -85,B 0,C 180,E1 -24795.007,E2 -24795.007} C_VEL
LIN {X 0,Y 133.454,Z 296.815,A -85,B 0,C 180,E1 -24797.499,E2 -24797.499} C_VEL
LIN {X 0,Y 134.197,Z 299.112,A -85,B 0,C 180,E1 -24801.772,E2 -24801.772} C_VEL
LIN {X 0,Y 135.613,Z 300.37,A -85,B 0,C 180,E1 -24806.014,E2 -24806.014} C_VEL
LIN {X 0,Y 137.7,Z 300.612,A -85,B 0,C 180,E1 -24810.187,E2 -24810.187} C_VEL
LIN {X 0,Y 140.487,Z 299.825,A -85,B 0,C 180,E1 -24814.218,E2 -24814.218} C_VEL
LIN {X 0,Y 143.884,Z 297.993,A -85,B 0,C 180,E1 -24818.132,E2 -24818.132} C_VEL
LIN {X 0,Y 147.953,Z 295.048,A -85,B 0,C 180,E1 -24821.81,E2 -24821.81} C_VEL
LIN {X 0,Y 152.579,Z 290.754,A -85,B 0,C 180,E1 -24825.304,E2 -24825.304} C_VEL
LIN {X 0,Y 156.27,Z 286.849,A -85,B 0,C 180,E1 -24827.663,E2 -24827.663} C_VEL
LIN {X 0,Y 157.56,Z 284.793,A -85,B 0,C 180,E1 -24828.906,E2 -24828.906} C_VEL
LIN {X 0,Y 158.849,Z 281.437,A -85,B 0,C 180,E1 -24831.094,E2 -24831.094} C_VEL
LIN {X 0,Y 159.875,Z 277.488,A -85,B 0,C 180,E1 -24833.693,E2 -24833.693} C_VEL
LIN {X 0,Y 160.31,Z 273.673,A -85,B 0,C 180,E1 -24836.232,E2 -24836.232} C_VEL
LIN {X 0,Y 159.957,Z 268.758,A -85,B 0,C 180,E1 -24840.002,E2 -24840.002} C_VEL
LIN {X 0,Y 159.172,Z 264.479,A -85,B 0,C 180,E1 -24843.8,E2 -24843.8} C_VEL
LIN {X 0,Y 158.851,Z 263.296,A -85,B 0,C 180,E1 -24845.079,E2 -24845.079} C_VEL
LIN {X 0,Y 157.309,Z 259.407,A -85,B 0,C 180,E1 -24850.619,E2 -24850.619} C_VEL
LIN {X 0,Y 155.691,Z 257.331,A -85,B 0,C 180,E1 -24858.568,E2 -24858.568} C_VEL
LIN {X 0,Y 155.606,Z 257.195,A -85,B 0,C 180,E1 -24861.184,E2 -24861.184} C_VEL
LIN {X 0,Y 155.69,Z 258.147,A -85,B 0,C 180,E1 -24865.47,E2 -24865.47} C_VEL
LIN {X 0,Y 156.863,Z 261.83,A -85,B 0,C 180,E1 -24872.526,E2 -24872.526} C_VEL
LIN {X 0,Y 157.288,Z 262.974,A -85,B 0,C 180,E1 -24873.996,E2 -24873.996} C_VEL
LIN {X 0,Y 158.465,Z 268.232,A -85,B 0,C 180,E1 -24879.109,E2 -24879.109} C_VEL
LIN {X 0,Y 159.16,Z 271.107,A -85,B 0,C 180,E1 -24881.482,E2 -24881.482} C_VEL
LIN {X 0,Y 159.957,Z 276.4,A -85,B 0,C 180,E1 -24885.333,E2 -24885.333} C_VEL
LIN {X 0,Y 160.21,Z 279.749,A -85,B 0,C 180,E1 -24887.457,E2 -24887.457} C_VEL
LIN {X 0,Y 158.355,Z 285.665,A -85,B 0,C 180,E1 -24890.341,E2 -24890.341} C_VEL
LIN {X 0,Y 155.272,Z 292.608,A -85,B 0,C 180,E1 -24893.956,E2 -24893.956} C_VEL
LIN {X 0,Y 152.71,Z 296.946,A -85,B 0,C 180,E1 -24896.478,E2 -24896.478} C_VEL
LIN {X 0,Y 149.653,Z 300.668,A -85,B 0,C 180,E1 -24898.897,E2 -24898.897} C_VEL
LIN {X 0,Y 144.97,Z 305.146,A -85,B 0,C 180,E1 -24902.578,E2 -24902.578} C_VEL
LIN {X 0,Y 140.99,Z 308.35,A -85,B 0,C 180,E1 -24906.499,E2 -24906.499} C_VEL
LIN {X 0,Y 138.795,Z 309.909,A -85,B 0,C 180,E1 -24909.241,E2 -24909.241} C_VEL
LIN {X 0,Y 137.075,Z 310.955,A -85,B 0,C 180,E1 -24912.084,E2 -24912.084} C_VEL
LIN {X 0,Y 135.708,Z 311.459,A -85,B 0,C 180,E1 -24914.993,E2 -24914.993} C_VEL
LIN {X 0,Y 134.694,Z 311.534,A -85,B 0,C 180,E1 -24917.954,E2 -24917.954} C_VEL
LIN {X 0,Y 134.035,Z 311.184,A -85,B 0,C 180,E1 -24920.95,E2 -24920.95} C_VEL
LIN {X 0,Y 133.768,Z 310.364,A -85,B 0,C 180,E1 -24923.969,E2 -24923.969} C_VEL
LIN {X 0,Y 133.855,Z 308.963,A -85,B 0,C 180,E1 -24926.991,E2 -24926.991} C_VEL
LIN {X 0,Y 134.064,Z 305.923,A -85,B 0,C 180,E1 -24931.503,E2 -24931.503} C_VEL
LIN {X 0,Y 134.007,Z 301.274,A -85,B 0,C 180,E1 -24936.021,E2 -24936.021} C_VEL
LIN {X 0,Y 134.449,Z 296.192,A -85,B 0,C 180,E1 -24939.782,E2 -24939.782} C_VEL
LIN {X 0,Y 135.062,Z 291.162,A -85,B 0,C 180,E1 -24942.777,E2 -24942.777} C_VEL
LIN {X 0,Y 135.969,Z 285.078,A -85,B 0,C 180,E1 -24945.746,E2 -24945.746} C_VEL
LIN {X 0,Y 137.252,Z 277.692,A -85,B 0,C 180,E1 -24948.665,E2 -24948.665} C_VEL
LIN {X 0,Y 137.332,Z 268.879,A -85,B 0,C 180,E1 -24951.508,E2 -24951.508} C_VEL
LIN {X 0,Y 137.07,Z 259.031,A -85,B 0,C 180,E1 -24953.998,E2 -24953.998} C_VEL
LIN {X 0,Y 136.754,Z 249.445,A -85,B 0,C 180,E1 -24955.902,E2 -24955.902} C_VEL
LIN {X 0,Y 136.213,Z 239.267,A -85,B 0,C 180,E1 -24957.461,E2 -24957.461} C_VEL
LIN {X 0,Y 135.968,Z 234.587,A -85,B 0,C 180,E1 -24958.043,E2 -24958.043} C_VEL
LIN {X 0,Y 137.264,Z 231.279,A -85,B 0,C 180,E1 -24962.522,E2 -24962.522} C_VEL
LIN {X 0,Y 137.418,Z 229.453,A -85,B 0,C 180,E1 -24965.082,E2 -24965.082} C_VEL
LIN {X 0,Y 136.752,Z 226.409,A -85,B 0,C 180,E1 -24969.564,E2 -24969.564} C_VEL
LIN {X 0,Y 136.39,Z 224.308,A -85,B 0,C 180,E1 -24972.915,E2 -24972.915} C_VEL
LIN {X 0,Y 136.068,Z 224.344,A -85,B 0,C 180,E1 -24977.817,E2 -24977.817} C_VEL
LIN {X 0,Y 136.031,Z 224.353,A -85,B 0,C 180,E1 -24981.683,E2 -24981.683} C_VEL
LIN {X 0,Y 136.089,Z 224.34,A -85,B 0,C 180,E1 -24985.72,E2 -24985.72} C_VEL
LIN {X 0,Y 136.149,Z 224.333,A -85,B 0,C 180,E1 -24992.314,E2 -24992.314} C_VEL
LIN {X 0,Y 136.246,Z 224.325,A -85,B 0,C 180,E1 -24998.831,E2 -24998.831} C_VEL
LIN {X 0,Y 136.272,Z 224.322,A -85,B 0,C 180,E1 -25005.054,E2 -25005.054} C_VEL
LIN {X 0,Y 136.273,Z 224.319,A -85,B 0,C 180,E1 -25005.497,E2 -25005.497} C_VEL
LIN {X 0,Y 135.631,Z 224.401,A -85,B 0,C 180,E1 -25007.967,E2 -25007.967} C_VEL
LIN {X 0,Y 134.09,Z 224.593,A -85,B 0,C 180,E1 -25010.406,E2 -25010.406} C_VEL
LIN {X 0,Y 130.617,Z 225.027,A -85,B 0,C 180,E1 -25015.399,E2 -25015.399} C_VEL
LIN {X 0,Y 129.857,Z 225.115,A -85,B 0,C 180,E1 -25018.022,E2 -25018.022} C_VEL
LIN {X 0,Y 129.901,Z 225.108,A -85,B 0,C 180,E1 -25018.906,E2 -25018.906} C_VEL
LIN {X 0,Y 130.09,Z 225.09,A -85,B 0,C 180,E1 -25019.997,E2 -25019.997} C_VEL
LIN {X 0,Y 129.474,Z 225.169,A -85,B 0,C 180,E1 -25029.369,E2 -25029.369} C_VEL
LIN {X 0,Y 129.3,Z 225.191,A -85,B 0,C 180,E1 -25032.554,E2 -25032.554} C_VEL
LIN {X 0,Y 129.114,Z 225.215,A -85,B 0,C 180,E1 -25039.059,E2 -25039.059} C_VEL
LIN {X 0,Y 129.106,Z 225.211,A -85,B 0,C 180,E1 -25042.396,E2 -25042.396} C_VEL
LIN {X 0,Y 129.035,Z 225.222,A -85,B 0,C 180,E1 -25049.37,E2 -25049.37} C_VEL
LIN {X 0,Y 128.99,Z 225.229,A -85,B 0,C 180,E1 -25055.186,E2 -25055.186} C_VEL
LIN {X 0,Y 128.948,Z 225.231,A -85,B 0,C 180,E1 -25060.842,E2 -25060.842} C_VEL
LIN {X 0,Y 128.918,Z 225.238,A -85,B 0,C 180,E1 -25065.125,E2 -25065.125} C_VEL
LIN {X 0,Y 128.938,Z 225.232,A -85,B 0,C 180,E1 -25069.733,E2 -25069.733} C_VEL
LIN {X 0,Y 128.955,Z 225.232,A -85,B 0,C 180,E1 -25074.829,E2 -25074.829} C_VEL
LIN {X 0,Y 129.046,Z 225.222,A -85,B 0,C 180,E1 -25080.649,E2 -25080.649} C_VEL
LIN {X 0,Y 129.102,Z 225.216,A -85,B 0,C 180,E1 -25087.726,E2 -25087.726} C_VEL
LIN {X 0,Y 129.149,Z 225.21,A -85,B 0,C 180,E1 -25090.943,E2 -25090.943} C_VEL
LIN {X 0,Y 129.41,Z 225.177,A -85,B 0,C 180,E1 -25097.819,E2 -25097.819} C_VEL
LIN {X 0,Y 129.511,Z 225.161,A -85,B 0,C 180,E1 -25100.63,E2 -25100.63} C_VEL
LIN {X 0,Y 130.082,Z 225.088,A -85,B 0,C 180,E1 -25109.999,E2 -25109.999} C_VEL
LIN {X 0,Y 129.46,Z 225.171,A -85,B 0,C 180,E1 -25116.233,E2 -25116.233} C_VEL
LIN {X 0,Y 129.367,Z 225.178,A -85,B 0,C 180,E1 -25119.379,E2 -25119.379} C_VEL
LIN {X 0,Y 128.952,Z 225.235,A -85,B 0,C 180,E1 -25122.591,E2 -25122.591} C_VEL
LIN {X 0,Y 128.221,Z 225.504,A -85,B 0,C 180,E1 -25127.134,E2 -25127.134} C_VEL
LIN {X 0,Y 129.873,Z 236.48,A -85,B 0,C 180,E1 -25128.946,E2 -25128.946} C_VEL
LIN {X 0,Y 130.969,Z 245.401,A -85,B 0,C 180,E1 -25130.824,E2 -25130.824} C_VEL
LIN {X 0,Y 131.861,Z 254.375,A -85,B 0,C 180,E1 -25133.146,E2 -25133.146} C_VEL
LIN {X 0,Y 132.059,Z 258.478,A -85,B 0,C 180,E1 -25134.358,E2 -25134.358} C_VEL
LIN {X 0,Y 130.625,Z 265.873,A -85,B 0,C 180,E1 -25136.782,E2 -25136.782} C_VEL
LIN {X 0,Y 129.347,Z 272.864,A -85,B 0,C 180,E1 -25139.623,E2 -25139.623} C_VEL
LIN {X 0,Y 128.38,Z 278.309,A -85,B 0,C 180,E1 -25142.298,E2 -25142.298} C_VEL
LIN {X 0,Y 127.35,Z 284.165,A -85,B 0,C 180,E1 -25145.811,E2 -25145.811} C_VEL
LIN {X 0,Y 126.689,Z 288.555,A -85,B 0,C 180,E1 -25149.051,E2 -25149.051} C_VEL
LIN {X 0,Y 126.251,Z 293.46,A -85,B 0,C 180,E1 -25153.646,E2 -25153.646} C_VEL
LIN {X 0,Y 126.429,Z 297.011,A -85,B 0,C 180,E1 -25158.164,E2 -25158.164} C_VEL
LIN {X 0,Y 127.265,Z 299.361,A -85,B 0,C 180,E1 -25162.598,E2 -25162.598} C_VEL
LIN {X 0,Y 128.786,Z 300.668,A -85,B 0,C 180,E1 -25166.93,E2 -25166.93} C_VEL
LIN {X 0,Y 130.944,Z 301.016,A -85,B 0,C 180,E1 -25171.119,E2 -25171.119} C_VEL
LIN {X 0,Y 133.774,Z 300.424,A -85,B 0,C 180,E1 -25175.15,E2 -25175.15} C_VEL
LIN {X 0,Y 137.113,Z 298.911,A -85,B 0,C 180,E1 -25178.976,E2 -25178.976} C_VEL
LIN {X 0,Y 141.131,Z 296.397,A -85,B 0,C 180,E1 -25182.618,E2 -25182.618} C_VEL
LIN {X 0,Y 145.665,Z 292.83,A -85,B 0,C 180,E1 -25186.043,E2 -25186.043} C_VEL
LIN {X 0,Y 150.714,Z 288.072,A -85,B 0,C 180,E1 -25189.252,E2 -25189.252} C_VEL
LIN {X 0,Y 151.936,Z 285.996,A -85,B 0,C 180,E1 -25190.685,E2 -25190.685} C_VEL
LIN {X 0,Y 153.494,Z 282.253,A -85,B 0,C 180,E1 -25193.429,E2 -25193.429} C_VEL
LIN {X 0,Y 154.465,Z 278.658,A -85,B 0,C 180,E1 -25196.089,E2 -25196.089} C_VEL
LIN {X 0,Y 154.753,Z 275.369,A -85,B 0,C 180,E1 -25198.7,E2 -25198.7} C_VEL
LIN {X 0,Y 154.544,Z 271.118,A -85,B 0,C 180,E1 -25202.609,E2 -25202.609} C_VEL
LIN {X 0,Y 154.228,Z 268.747,A -85,B 0,C 180,E1 -25205.231,E2 -25205.231} C_VEL
LIN {X 0,Y 153.165,Z 265.179,A -85,B 0,C 180,E1 -25210.578,E2 -25210.578} C_VEL
LIN {X 0,Y 151.838,Z 263.276,A -85,B 0,C 180,E1 -25218.907,E2 -25218.907} C_VEL
LIN {X 0,Y 151.783,Z 263.361,A -85,B 0,C 180,E1 -25222.172,E2 -25222.172} C_VEL
LIN {X 0,Y 151.824,Z 263.878,A -85,B 0,C 180,E1 -25224.623,E2 -25224.623} C_VEL
LIN {X 0,Y 152.295,Z 266.482,A -85,B 0,C 180,E1 -25230.508,E2 -25230.508} C_VEL
LIN {X 0,Y 152.865,Z 268.365,A -85,B 0,C 180,E1 -25233.486,E2 -25233.486} C_VEL
LIN {X 0,Y 153.572,Z 272.514,A -85,B 0,C 180,E1 -25237.937,E2 -25237.937} C_VEL
LIN {X 0,Y 154.047,Z 276.59,A -85,B 0,C 180,E1 -25241.554,E2 -25241.554} C_VEL
LIN {X 0,Y 154.499,Z 281.691,A -85,B 0,C 180,E1 -25245.624,E2 -25245.624} C_VEL
LIN {X 0,Y 154.204,Z 283.676,A -85,B 0,C 180,E1 -25246.872,E2 -25246.872} C_VEL
LIN {X 0,Y 152.013,Z 288.874,A -85,B 0,C 180,E1 -25249.665,E2 -25249.665} C_VEL
LIN {X 0,Y 149.539,Z 293.5,A -85,B 0,C 180,E1 -25252.341,E2 -25252.341} C_VEL
LIN {X 0,Y 146.854,Z 297.613,A -85,B 0,C 180,E1 -25254.951,E2 -25254.951} C_VEL
LIN {X 0,Y 143.653,Z 301.207,A -85,B 0,C 180,E1 -25257.442,E2 -25257.442} C_VEL
LIN {X 0,Y 138.713,Z 305.412,A -85,B 0,C 180,E1 -25261.229,E2 -25261.229} C_VEL
LIN {X 0,Y 134.525,Z 308.422,A -85,B 0,C 180,E1 -25265.296,E2 -25265.296} C_VEL
LIN {X 0,Y 132.166,Z 309.809,A -85,B 0,C 180,E1 -25268.147,E2 -25268.147} C_VEL
LIN {X 0,Y 130.311,Z 310.766,A -85,B 0,C 180,E1 -25271.12,E2 -25271.12} C_VEL
LIN {X 0,Y 128.838,Z 311.202,A -85,B 0,C 180,E1 -25274.173,E2 -25274.173} C_VEL
LIN {X 0,Y 127.769,Z 311.121,A -85,B 0,C 180,E1 -25277.29,E2 -25277.29} C_VEL
LIN {X 0,Y 127.044,Z 310.614,A -85,B 0,C 180,E1 -25280.448,E2 -25280.448} C_VEL
LIN {X 0,Y 126.743,Z 309.676,A -85,B 0,C 180,E1 -25283.633,E2 -25283.633} C_VEL
LIN {X 0,Y 126.855,Z 307.366,A -85,B 0,C 180,E1 -25288.219,E2 -25288.219} C_VEL
LIN {X 0,Y 127.013,Z 304.946,A -85,B 0,C 180,E1 -25291.586,E2 -25291.586} C_VEL
LIN {X 0,Y 126.924,Z 302.086,A -85,B 0,C 180,E1 -25294.636,E2 -25294.636} C_VEL
LIN {X 0,Y 127.229,Z 297.11,A -85,B 0,C 180,E1 -25298.738,E2 -25298.738} C_VEL
LIN {X 0,Y 127.944,Z 290.954,A -85,B 0,C 180,E1 -25302.693,E2 -25302.693} C_VEL
LIN {X 0,Y 128.854,Z 284.894,A -85,B 0,C 180,E1 -25305.826,E2 -25305.826} C_VEL
LIN {X 0,Y 130.178,Z 277.544,A -85,B 0,C 180,E1 -25308.901,E2 -25308.901} C_VEL
LIN {X 0,Y 130.274,Z 269.168,A -85,B 0,C 180,E1 -25311.771,E2 -25311.771} C_VEL
LIN {X 0,Y 130.046,Z 258.487,A -85,B 0,C 180,E1 -25314.643,E2 -25314.643} C_VEL
LIN {X 0,Y 129.778,Z 249.487,A -85,B 0,C 180,E1 -25316.537,E2 -25316.537} C_VEL
LIN {X 0,Y 129.3,Z 239.846,A -85,B 0,C 180,E1 -25318.123,E2 -25318.123} C_VEL
LIN {X 0,Y 129.08,Z 234.291,A -85,B 0,C 180,E1 -25318.896,E2 -25318.896} C_VEL
LIN {X 0,Y 130.154,Z 231.665,A -85,B 0,C 180,E1 -25322.683,E2 -25322.683} C_VEL
LIN {X 0,Y 130.417,Z 230.616,A -85,B 0,C 180,E1 -25324.211,E2 -25324.211} C_VEL
LIN {X 0,Y 129.548,Z 226.488,A -85,B 0,C 180,E1 -25330.618,E2 -25330.618} C_VEL
LIN {X 0,Y 129.323,Z 225.188,A -85,B 0,C 180,E1 -25332.823,E2 -25332.823} C_VEL
LIN {X 0,Y 128.983,Z 225.23,A -85,B 0,C 180,E1 -25339.715,E2 -25339.715} C_VEL
LIN {X 0,Y 128.985,Z 225.224,A -85,B 0,C 180,E1 -25344.817,E2 -25344.817} C_VEL
LIN {X 0,Y 129.021,Z 225.224,A -85,B 0,C 180,E1 -25350.641,E2 -25350.641} C_VEL
LIN {X 0,Y 129.032,Z 225.22,A -85,B 0,C 180,E1 -25354.165,E2 -25354.165} C_VEL
LIN {X 0,Y 129.111,Z 225.216,A -85,B 0,C 180,E1 -25357.726,E2 -25357.726} C_VEL
LIN {X 0,Y 129.156,Z 225.204,A -85,B 0,C 180,E1 -25360.942,E2 -25360.942} C_VEL
LIN {X 0,Y 129.37,Z 225.18,A -85,B 0,C 180,E1 -25367.92,E2 -25367.92} C_VEL
LIN {X 0,Y 129.48,Z 225.163,A -85,B 0,C 180,E1 -25370.626,E2 -25370.626} C_VEL
LIN {X 0,Y 129.901,Z 225.108,A -85,B 0,C 180,E1 -25378.906,E2 -25378.906} C_VEL
LIN {X 0,Y 129.773,Z 225.13,A -85,B 0,C 180,E1 -25380.627,E2 -25380.627} C_VEL
LIN {X 0,Y 128.501,Z 225.293,A -85,B 0,C 180,E1 -25383.18,E2 -25383.18} C_VEL
LIN {X 0,Y 125.067,Z 225.724,A -85,B 0,C 180,E1 -25387.44,E2 -25387.44} C_VEL
LIN {X 0,Y 122.398,Z 226.05,A -85,B 0,C 180,E1 -25391.989,E2 -25391.989} C_VEL
LIN {X 0,Y 122.222,Z 226.07,A -85,B 0,C 180,E1 -25392.938,E2 -25392.938} C_VEL
LIN {X 0,Y 122.076,Z 226.088,A -85,B 0,C 180,E1 -25396.726,E2 -25396.726} C_VEL
LIN {X 0,Y 122.021,Z 226.091,A -85,B 0,C 180,E1 -25402.845,E2 -25402.845} C_VEL
LIN {X 0,Y 121.955,Z 226.106,A -85,B 0,C 180,E1 -25407.45,E2 -25407.45} C_VEL
LIN {X 0,Y 121.91,Z 226.105,A -85,B 0,C 180,E1 -25411.251,E2 -25411.251} C_VEL
LIN {X 0,Y 121.91,Z 226.113,A -85,B 0,C 180,E1 -25416.187,E2 -25416.187} C_VEL
LIN {X 0,Y 121.881,Z 226.111,A -85,B 0,C 180,E1 -25421.442,E2 -25421.442} C_VEL
LIN {X 0,Y 121.868,Z 226.111,A -85,B 0,C 180,E1 -25428.559,E2 -25428.559} C_VEL
LIN {X 0,Y 121.906,Z 226.11,A -85,B 0,C 180,E1 -25434.794,E2 -25434.794} C_VEL
LIN {X 0,Y 121.934,Z 226.109,A -85,B 0,C 180,E1 -25439.826,E2 -25439.826} C_VEL
LIN {X 0,Y 121.978,Z 226.099,A -85,B 0,C 180,E1 -25446.213,E2 -25446.213} C_VEL
LIN {X 0,Y 122.041,Z 226.095,A -85,B 0,C 180,E1 -25449.786,E2 -25449.786} C_VEL
LIN {X 0,Y 122.357,Z 226.056,A -85,B 0,C 180,E1 -25457.525,E2 -25457.525} C_VEL
LIN {X 0,Y 122.441,Z 226.043,A -85,B 0,C 180,E1 -25460.084,E2 -25460.084} C_VEL
LIN {X 0,Y 122.6,Z 226.027,A -85,B 0,C 180,E1 -25466.713,E2 -25466.713} C_VEL
LIN {X 0,Y 123.036,Z 225.965,A -85,B 0,C 180,E1 -25469.999,E2 -25469.999} C_VEL
LIN {X 0,Y 122.389,Z 226.05,A -85,B 0,C 180,E1 -25476.594,E2 -25476.594} C_VEL
LIN {X 0,Y 122.049,Z 226.094,A -85,B 0,C 180,E1 -25481.802,E2 -25481.802} C_VEL
LIN {X 0,Y 121.318,Z 226.183,A -85,B 0,C 180,E1 -25486.295,E2 -25486.295} C_VEL
LIN {X 0,Y 122.942,Z 237.401,A -85,B 0,C 180,E1 -25488.324,E2 -25488.324} C_VEL
LIN {X 0,Y 124.002,Z 246.189,A -85,B 0,C 180,E1 -25490.312,E2 -25490.312} C_VEL
LIN {X 0,Y 124.848,Z 255.109,A -85,B 0,C 180,E1 -25492.768,E2 -25492.768} C_VEL
LIN {X 0,Y 125.083,Z 257.865,A -85,B 0,C 180,E1 -25493.613,E2 -25493.613} C_VEL
LIN {X 0,Y 123.499,Z 266.414,A -85,B 0,C 180,E1 -25496.584,E2 -25496.584} C_VEL
LIN {X 0,Y 122.308,Z 272.641,A -85,B 0,C 180,E1 -25499.236,E2 -25499.236} C_VEL
LIN {X 0,Y 121.15,Z 278.842,A -85,B 0,C 180,E1 -25502.452,E2 -25502.452} C_VEL
LIN {X 0,Y 120.252,Z 284.083,A -85,B 0,C 180,E1 -25505.763,E2 -25505.763} C_VEL
LIN {X 0,Y 119.611,Z 288.325,A -85,B 0,C 180,E1 -25509,E2 -25509} C_VEL
LIN {X 0,Y 119.192,Z 292.223,A -85,B 0,C 180,E1 -25512.643,E2 -25512.643} C_VEL
LIN {X 0,Y 119.156,Z 294.423,A -85,B 0,C 180,E1 -25515.054,E2 -25515.054} C_VEL
LIN {X 0,Y 119.546,Z 297.744,A -85,B 0,C 180,E1 -25519.84,E2 -25519.84} C_VEL
LIN {X 0,Y 120.709,Z 299.945,A -85,B 0,C 180,E1 -25524.598,E2 -25524.598} C_VEL
LIN {X 0,Y 122.628,Z 301.136,A -85,B 0,C 180,E1 -25529.279,E2 -25529.279} C_VEL
LIN {X 0,Y 125.33,Z 301.318,A -85,B 0,C 180,E1 -25533.793,E2 -25533.793} C_VEL
LIN {X 0,Y 128.742,Z 300.486,A -85,B 0,C 180,E1 -25538.128,E2 -25538.128} C_VEL
LIN {X 0,Y 132.856,Z 298.623,A -85,B 0,C 180,E1 -25542.21,E2 -25542.21} C_VEL
LIN {X 0,Y 137.598,Z 295.638,A -85,B 0,C 180,E1 -25546.036,E2 -25546.036} C_VEL
LIN {X 0,Y 142.923,Z 291.371,A -85,B 0,C 180,E1 -25549.565,E2 -25549.565} C_VEL
LIN {X 0,Y 144.808,Z 289.687,A -85,B 0,C 180,E1 -25550.668,E2 -25550.668} C_VEL
LIN {X 0,Y 146.796,Z 286.589,A -85,B 0,C 180,E1 -25553.128,E2 -25553.128} C_VEL
LIN {X 0,Y 148.422,Z 282.67,A -85,B 0,C 180,E1 -25556.367,E2 -25556.367} C_VEL
LIN {X 0,Y 149.087,Z 280.093,A -85,B 0,C 180,E1 -25558.652,E2 -25558.652} C_VEL
LIN {X 0,Y 149.28,Z 276.088,A -85,B 0,C 180,E1 -25562.701,E2 -25562.701} C_VEL
LIN {X 0,Y 149.259,Z 273.881,A -85,B 0,C 180,E1 -25565.406,E2 -25565.406} C_VEL
LIN {X 0,Y 148.557,Z 270.558,A -85,B 0,C 180,E1 -25570.91,E2 -25570.91} C_VEL
LIN {X 0,Y 147.579,Z 269.14,A -85,B 0,C 180,E1 -25577.743,E2 -25577.743} C_VEL
LIN {X 0,Y 147.547,Z 268.952,A -85,B 0,C 180,E1 -25579.479,E2 -25579.479} C_VEL
LIN {X 0,Y 147.52,Z 269.115,A -85,B 0,C 180,E1 -25582.406,E2 -25582.406} C_VEL
LIN {X 0,Y 147.507,Z 269.879,A -85,B 0,C 180,E1 -25585.394,E2 -25585.394} C_VEL
LIN {X 0,Y 147.913,Z 272.675,A -85,B 0,C 180,E1 -25591.513,E2 -25591.513} C_VEL
LIN {X 0,Y 148.145,Z 273.572,A -85,B 0,C 180,E1 -25593.065,E2 -25593.065} C_VEL
LIN {X 0,Y 148.515,Z 277.856,A -85,B 0,C 180,E1 -25597.968,E2 -25597.968} C_VEL
LIN {X 0,Y 148.693,Z 282.575,A -85,B 0,C 180,E1 -25602.504,E2 -25602.504} C_VEL
LIN {X 0,Y 148.614,Z 285.761,A -85,B 0,C 180,E1 -25605.185,E2 -25605.185} C_VEL
LIN {X 0,Y 147.387,Z 288.65,A -85,B 0,C 180,E1 -25607.014,E2 -25607.014} C_VEL
LIN {X 0,Y 143.962,Z 294.485,A -85,B 0,C 180,E1 -25610.607,E2 -25610.607} C_VEL
LIN {X 0,Y 141.066,Z 298.319,A -85,B 0,C 180,E1 -25613.285,E2 -25613.285} C_VEL
LIN {X 0,Y 137.752,Z 301.666,A -85,B 0,C 180,E1 -25615.861,E2 -25615.861} C_VEL
LIN {X 0,Y 132.546,Z 305.681,A -85,B 0,C 180,E1 -25619.754,E2 -25619.754} C_VEL
LIN {X 0,Y 128.1,Z 308.514,A -85,B 0,C 180,E1 -25623.966,E2 -25623.966} C_VEL
LIN {X 0,Y 125.597,Z 309.728,A -85,B 0,C 180,E1 -25626.94,E2 -25626.94} C_VEL
LIN {X 0,Y 123.59,Z 310.513,A -85,B 0,C 180,E1 -25630.051,E2 -25630.051} C_VEL
LIN {X 0,Y 122.001,Z 310.878,A -85,B 0,C 180,E1 -25633.26,E2 -25633.26} C_VEL
LIN {X 0,Y 120.834,Z 310.708,A -85,B 0,C 180,E1 -25636.547,E2 -25636.547} C_VEL
LIN {X 0,Y 120.073,Z 310.046,A -85,B 0,C 180,E1 -25639.887,E2 -25639.887} C_VEL
LIN {X 0,Y 119.735,Z 307.614,A -85,B 0,C 180,E1 -25646.269,E2 -25646.269} C_VEL
LIN {X 0,Y 119.961,Z 305.276,A -85,B 0,C 180,E1 -25650.001,E2 -25650.001} C_VEL
LIN {X 0,Y 119.878,Z 301.129,A -85,B 0,C 180,E1 -25654.665,E2 -25654.665} C_VEL
LIN {X 0,Y 120.26,Z 295.686,A -85,B 0,C 180,E1 -25659.249,E2 -25659.249} C_VEL
LIN {X 0,Y 121.032,Z 289.322,A -85,B 0,C 180,E1 -25663.431,E2 -25663.431} C_VEL
LIN {X 0,Y 122.362,Z 281.317,A -85,B 0,C 180,E1 -25667.551,E2 -25667.551} C_VEL
LIN {X 0,Y 123.215,Z 276.374,A -85,B 0,C 180,E1 -25669.579,E2 -25669.579} C_VEL
LIN {X 0,Y 123.167,Z 266.145,A -85,B 0,C 180,E1 -25673.098,E2 -25673.098} C_VEL
LIN {X 0,Y 123.018,Z 257.676,A -85,B 0,C 180,E1 -25675.409,E2 -25675.409} C_VEL
LIN {X 0,Y 122.766,Z 248.166,A -85,B 0,C 180,E1 -25677.481,E2 -25677.481} C_VEL
LIN {X 0,Y 122.282,Z 237.235,A -85,B 0,C 180,E1 -25679.301,E2 -25679.301} C_VEL
LIN {X 0,Y 122.134,Z 234.023,A -85,B 0,C 180,E1 -25679.8,E2 -25679.8} C_VEL
LIN {X 0,Y 123.042,Z 232.001,A -85,B 0,C 180,E1 -25682.864,E2 -25682.864} C_VEL
LIN {X 0,Y 123.251,Z 230.781,A -85,B 0,C 180,E1 -25684.766,E2 -25684.766} C_VEL
LIN {X 0,Y 122.41,Z 226.576,A -85,B 0,C 180,E1 -25691.719,E2 -25691.719} C_VEL
LIN {X 0,Y 122.272,Z 226.067,A -85,B 0,C 180,E1 -25692.827,E2 -25692.827} C_VEL
LIN {X 0,Y 121.888,Z 226.115,A -85,B 0,C 180,E1 -25700.632,E2 -25700.632} C_VEL
LIN {X 0,Y 121.937,Z 226.101,A -85,B 0,C 180,E1 -25704.802,E2 -25704.802} C_VEL
LIN {X 0,Y 121.933,Z 226.11,A -85,B 0,C 180,E1 -25709.835,E2 -25709.835} C_VEL
LIN {X 0,Y 121.987,Z 226.102,A -85,B 0,C 180,E1 -25716.213,E2 -25716.213} C_VEL
LIN {X 0,Y 122.049,Z 226.091,A -85,B 0,C 180,E1 -25719.785,E2 -25719.785} C_VEL
LIN {X 0,Y 122.243,Z 226.07,A -85,B 0,C 180,E1 -25726.702,E2 -25726.702} C_VEL
LIN {X 0,Y 122.41,Z 226.043,A -85,B 0,C 180,E1 -25730.079,E2 -25730.079} C_VEL
LIN {X 0,Y 122.6,Z 226.024,A -85,B 0,C 180,E1 -25736.711,E2 -25736.711} C_VEL
LIN {X 0,Y 123.044,Z 225.968,A -85,B 0,C 180,E1 -25739.997,E2 -25739.997} C_VEL
LIN {X 0,Y 122.407,Z 226.042,A -85,B 0,C 180,E1 -25746.881,E2 -25746.881} C_VEL
LIN {X 0,Y 122.289,Z 226.064,A -85,B 0,C 180,E1 -25752.31,E2 -25752.31} C_VEL
LIN {X 0,Y 122.222,Z 226.07,A -85,B 0,C 180,E1 -25752.938,E2 -25752.938} C_VEL
LIN {X 0,Y 121.345,Z 226.178,A -85,B 0,C 180,E1 -25755.685,E2 -25755.685} C_VEL
LIN {X 0,Y 119.646,Z 226.394,A -85,B 0,C 180,E1 -25758.395,E2 -25758.395} C_VEL
LIN {X 0,Y 115.083,Z 226.96,A -85,B 0,C 180,E1 -25765.925,E2 -25765.925} C_VEL
LIN {X 0,Y 114.809,Z 226.987,A -85,B 0,C 180,E1 -25767.923,E2 -25767.923} C_VEL
LIN {X 0,Y 114.836,Z 226.99,A -85,B 0,C 180,E1 -25773.418,E2 -25773.418} C_VEL
LIN {X 0,Y 114.8,Z 226.997,A -85,B 0,C 180,E1 -25777.744,E2 -25777.744} C_VEL
LIN {X 0,Y 114.792,Z 226.998,A -85,B 0,C 180,E1 -25782.718,E2 -25782.718} C_VEL
LIN {X 0,Y 114.791,Z 226.993,A -85,B 0,C 180,E1 -25787.664,E2 -25787.664} C_VEL
LIN {X 0,Y 114.784,Z 226.999,A -85,B 0,C 180,E1 -25792.741,E2 -25792.741} C_VEL
LIN {X 0,Y 114.857,Z 226.988,A -85,B 0,C 180,E1 -25798.936,E2 -25798.936} C_VEL
LIN {X 0,Y 114.941,Z 226.976,A -85,B 0,C 180,E1 -25806.506,E2 -25806.506} C_VEL
LIN {X 0,Y 115.008,Z 226.967,A -85,B 0,C 180,E1 -25812.208,E2 -25812.208} C_VEL
LIN {X 0,Y 115.278,Z 226.939,A -85,B 0,C 180,E1 -25817.261,E2 -25817.261} C_VEL
LIN {X 0,Y 115.382,Z 226.92,A -85,B 0,C 180,E1 -25823.002,E2 -25823.002} C_VEL
LIN {X 0,Y 115.987,Z 226.843,A -85,B 0,C 180,E1 -25829.999,E2 -25829.999} C_VEL
LIN {X 0,Y 115.312,Z 226.93,A -85,B 0,C 180,E1 -25837.001,E2 -25837.001} C_VEL
LIN {X 0,Y 114.94,Z 226.979,A -85,B 0,C 180,E1 -25841.969,E2 -25841.969} C_VEL
LIN {X 0,Y 114.412,Z 227.043,A -85,B 0,C 180,E1 -25845.361,E2 -25845.361} C_VEL
LIN {X 0,Y 116.052,Z 238.286,A -85,B 0,C 180,E1 -25847.625,E2 -25847.625} C_VEL
LIN {X 0,Y 117.048,Z 246.973,A -85,B 0,C 180,E1 -25849.739,E2 -25849.739} C_VEL
LIN {X 0,Y 117.975,Z 257.189,A -85,B 0,C 180,E1 -25852.781,E2 -25852.781} C_VEL
LIN {X 0,Y 117.461,Z 261.527,A -85,B 0,C 180,E1 -25854.289,E2 -25854.289} C_VEL
LIN {X 0,Y 115.769,Z 270.124,A -85,B 0,C 180,E1 -25857.705,E2 -25857.705} C_VEL
LIN {X 0,Y 114.349,Z 277.327,A -85,B 0,C 180,E1 -25861.364,E2 -25861.364} C_VEL
LIN {X 0,Y 113.053,Z 284.505,A -85,B 0,C 180,E1 -25866.091,E2 -25866.091} C_VEL
LIN {X 0,Y 112.369,Z 289.156,A -85,B 0,C 180,E1 -25869.952,E2 -25869.952} C_VEL
LIN {X 0,Y 112.091,Z 292.745,A -85,B 0,C 180,E1 -25873.605,E2 -25873.605} C_VEL
LIN {X 0,Y 112.106,Z 295.095,A -85,B 0,C 180,E1 -25876.407,E2 -25876.407} C_VEL
LIN {X 0,Y 112.731,Z 298.266,A -85,B 0,C 180,E1 -25881.437,E2 -25881.437} C_VEL
LIN {X 0,Y 114.124,Z 300.373,A -85,B 0,C 180,E1 -25886.346,E2 -25886.346} C_VEL
LIN {X 0,Y 116.26,Z 301.504,A -85,B 0,C 180,E1 -25891.083,E2 -25891.083} C_VEL
LIN {X 0,Y 119.169,Z 301.69,A -85,B 0,C 180,E1 -25895.621,E2 -25895.621} C_VEL
LIN {X 0,Y 122.723,Z 300.951,A -85,B 0,C 180,E1 -25899.907,E2 -25899.907} C_VEL
LIN {X 0,Y 126.938,Z 299.272,A -85,B 0,C 180,E1 -25903.932,E2 -25903.932} C_VEL
LIN {X 0,Y 131.732,Z 296.613,A -85,B 0,C 180,E1 -25907.681,E2 -25907.681} C_VEL
LIN {X 0,Y 137.146,Z 292.817,A -85,B 0,C 180,E1 -25911.159,E2 -25911.159} C_VEL
LIN {X 0,Y 139.552,Z 290.615,A -85,B 0,C 180,E1 -25912.77,E2 -25912.77} C_VEL
LIN {X 0,Y 141.127,Z 288.407,A -85,B 0,C 180,E1 -25914.858,E2 -25914.858} C_VEL
LIN {X 0,Y 142.437,Z 285.899,A -85,B 0,C 180,E1 -25917.174,E2 -25917.174} C_VEL
LIN {X 0,Y 143.349,Z 283.112,A -85,B 0,C 180,E1 -25920.002,E2 -25920.002} C_VEL
LIN {X 0,Y 143.912,Z 279.653,A -85,B 0,C 180,E1 -25924.203,E2 -25924.203} C_VEL
LIN {X 0,Y 143.925,Z 278.61,A -85,B 0,C 180,E1 -25925.607,E2 -25925.607} C_VEL
LIN {X 0,Y 143.533,Z 275.577,A -85,B 0,C 180,E1 -25931.684,E2 -25931.684} C_VEL
LIN {X 0,Y 142.913,Z 274.522,A -85,B 0,C 180,E1 -25937.164,E2 -25937.164} C_VEL
LIN {X 0,Y 142.814,Z 274.337,A -85,B 0,C 180,E1 -25940.772,E2 -25940.772} C_VEL
LIN {X 0,Y 142.801,Z 274.674,A -85,B 0,C 180,E1 -25943.189,E2 -25943.189} C_VEL
LIN {X 0,Y 142.767,Z 276.092,A -85,B 0,C 180,E1 -25947.615,E2 -25947.615} C_VEL
LIN {X 0,Y 143.139,Z 278.544,A -85,B 0,C 180,E1 -25952.692,E2 -25952.692} C_VEL
LIN {X 0,Y 143.101,Z 282.922,A -85,B 0,C 180,E1 -25958.206,E2 -25958.206} C_VEL
LIN {X 0,Y 142.813,Z 288.085,A -85,B 0,C 180,E1 -25963.55,E2 -25963.55} C_VEL
LIN {X 0,Y 142.484,Z 289.306,A -85,B 0,C 180,E1 -25964.546,E2 -25964.546} C_VEL
LIN {X 0,Y 139.912,Z 293.364,A -85,B 0,C 180,E1 -25967.303,E2 -25967.303} C_VEL
LIN {X 0,Y 136.39,Z 297.943,A -85,B 0,C 180,E1 -25970.621,E2 -25970.621} C_VEL
LIN {X 0,Y 133.775,Z 300.703,A -85,B 0,C 180,E1 -25972.832,E2 -25972.832} C_VEL
LIN {X 0,Y 130.043,Z 303.652,A -85,B 0,C 180,E1 -25975.427,E2 -25975.427} C_VEL
LIN {X 0,Y 124.817,Z 306.947,A -85,B 0,C 180,E1 -25979.552,E2 -25979.552} C_VEL
LIN {X 0,Y 121.756,Z 308.579,A -85,B 0,C 180,E1 -25982.499,E2 -25982.499} C_VEL
LIN {X 0,Y 119.094,Z 309.65,A -85,B 0,C 180,E1 -25985.602,E2 -25985.602} C_VEL
LIN {X 0,Y 116.919,Z 310.262,A -85,B 0,C 180,E1 -25988.86,E2 -25988.86} C_VEL
LIN {X 0,Y 115.205,Z 310.46,A -85,B 0,C 180,E1 -25992.241,E2 -25992.241} C_VEL
LIN {X 0,Y 113.932,Z 310.236,A -85,B 0,C 180,E1 -25995.716,E2 -25995.716} C_VEL
LIN {X 0,Y 113.096,Z 309.465,A -85,B 0,C 180,E1 -25999.256,E2 -25999.256} C_VEL
LIN {X 0,Y 112.719,Z 306.712,A -85,B 0,C 180,E1 -26006.064,E2 -26006.064} C_VEL
LIN {X 0,Y 112.921,Z 304.244,A -85,B 0,C 180,E1 -26010.001,E2 -26010.001} C_VEL
LIN {X 0,Y 112.838,Z 300.093,A -85,B 0,C 180,E1 -26014.735,E2 -26014.735} C_VEL
LIN {X 0,Y 113.163,Z 295.353,A -85,B 0,C 180,E1 -26018.933,E2 -26018.933} C_VEL
LIN {X 0,Y 113.733,Z 290.381,A -85,B 0,C 180,E1 -26022.491,E2 -26022.491} C_VEL
LIN {X 0,Y 114.675,Z 284.369,A -85,B 0,C 180,E1 -26026.01,E2 -26026.01} C_VEL
LIN {X 0,Y 116.032,Z 277.067,A -85,B 0,C 180,E1 -26029.46,E2 -26029.46} C_VEL
LIN {X 0,Y 116.135,Z 267.334,A -85,B 0,C 180,E1 -26033.164,E2 -26033.164} C_VEL
LIN {X 0,Y 116.014,Z 257.481,A -85,B 0,C 180,E1 -26036.053,E2 -26036.053} C_VEL
LIN {X 0,Y 115.819,Z 248.987,A -85,B 0,C 180,E1 -26038.053,E2 -26038.053} C_VEL
LIN {X 0,Y 115.444,Z 239.577,A -85,B 0,C 180,E1 -26039.795,E2 -26039.795} C_VEL
LIN {X 0,Y 115.242,Z 233.809,A -85,B 0,C 180,E1 -26040.694,E2 -26040.694} C_VEL
LIN {X 0,Y 115.942,Z 232.35,A -85,B 0,C 180,E1 -26043.063,E2 -26043.063} C_VEL
LIN {X 0,Y 116.113,Z 231.124,A -85,B 0,C 180,E1 -26045.101,E2 -26045.101} C_VEL
LIN {X 0,Y 115.261,Z 226.941,A -85,B 0,C 180,E1 -26052.491,E2 -26052.491} C_VEL
LIN {X 0,Y 114.882,Z 226.982,A -85,B 0,C 180,E1 -26057.703,E2 -26057.703} C_VEL
LIN {X 0,Y 114.811,Z 226.993,A -85,B 0,C 180,E1 -26062.73,E2 -26062.73} C_VEL
LIN {X 0,Y 114.867,Z 226.989,A -85,B 0,C 180,E1 -26068.936,E2 -26068.936} C_VEL
LIN {X 0,Y 114.951,Z 226.978,A -85,B 0,C 180,E1 -26076.506,E2 -26076.506} C_VEL
LIN {X 0,Y 115.015,Z 226.965,A -85,B 0,C 180,E1 -26082.207,E2 -26082.207} C_VEL
LIN {X 0,Y 115.256,Z 226.94,A -85,B 0,C 180,E1 -26087.331,E2 -26087.331} C_VEL
LIN {X 0,Y 115.368,Z 226.926,A -85,B 0,C 180,E1 -26092.999,E2 -26092.999} C_VEL
LIN {X 0,Y 115.995,Z 226.846,A -85,B 0,C 180,E1 -26099.997,E2 -26099.997} C_VEL
LIN {X 0,Y 115.365,Z 226.921,A -85,B 0,C 180,E1 -26106.995,E2 -26106.995} C_VEL
LIN {X 0,Y 115.185,Z 226.947,A -85,B 0,C 180,E1 -26112.795,E2 -26112.795} C_VEL
LIN {X 0,Y 114.984,Z 226.973,A -85,B 0,C 180,E1 -26117.791,E2 -26117.791} C_VEL
LIN {X 0,Y 114.944,Z 226.972,A -85,B 0,C 180,E1 -26123.486,E2 -26123.486} C_VEL
LIN {X 0,Y 114.809,Z 226.987,A -85,B 0,C 180,E1 -26127.923,E2 -26127.923} C_VEL
LIN {X 0,Y 114.511,Z 227.031,A -85,B 0,C 180,E1 -26129.88,E2 -26129.88} C_VEL
LIN {X 0,Y 113.688,Z 227.135,A -85,B 0,C 180,E1 -26131.813,E2 -26131.813} C_VEL
LIN {X 0,Y 111.207,Z 227.445,A -85,B 0,C 180,E1 -26135.665,E2 -26135.665} C_VEL
LIN {X 0,Y 107.911,Z 227.852,A -85,B 0,C 180,E1 -26141.794,E2 -26141.794} C_VEL
LIN {X 0,Y 107.67,Z 227.885,A -85,B 0,C 180,E1 -26143.938,E2 -26143.938} C_VEL
LIN {X 0,Y 107.684,Z 227.883,A -85,B 0,C 180,E1 -26151.547,E2 -26151.547} C_VEL
LIN {X 0,Y 107.792,Z 227.868,A -85,B 0,C 180,E1 -26158.56,E2 -26158.56} C_VEL
LIN {X 0,Y 107.905,Z 227.853,A -85,B 0,C 180,E1 -26166.996,E2 -26166.996} C_VEL
LIN {X 0,Y 108.032,Z 227.836,A -85,B 0,C 180,E1 -26174.916,E2 -26174.916} C_VEL
LIN {X 0,Y 108.282,Z 227.81,A -85,B 0,C 180,E1 -26178.771,E2 -26178.771} C_VEL
LIN {X 0,Y 108.451,Z 227.788,A -85,B 0,C 180,E1 -26186.284,E2 -26186.284} C_VEL
LIN {X 0,Y 108.936,Z 227.721,A -85,B 0,C 180,E1 -26189.999,E2 -26189.999} C_VEL
LIN {X 0,Y 108.23,Z 227.811,A -85,B 0,C 180,E1 -26197.462,E2 -26197.462} C_VEL
LIN {X 0,Y 107.831,Z 227.865,A -85,B 0,C 180,E1 -26202.158,E2 -26202.158} C_VEL
LIN {X 0,Y 107.483,Z 227.907,A -85,B 0,C 180,E1 -26204.504,E2 -26204.504} C_VEL
LIN {X 0,Y 108.895,Z 237.12,A -85,B 0,C 180,E1 -26206.4,E2 -26206.4} C_VEL
LIN {X 0,Y 109.923,Z 246.038,A -85,B 0,C 180,E1 -26208.643,E2 -26208.643} C_VEL
LIN {X 0,Y 110.722,Z 255.056,A -85,B 0,C 180,E1 -26211.405,E2 -26211.405} C_VEL
LIN {X 0,Y 110.928,Z 259.156,A -85,B 0,C 180,E1 -26212.833,E2 -26212.833} C_VEL
LIN {X 0,Y 109.171,Z 267.674,A -85,B 0,C 180,E1 -26216.221,E2 -26216.221} C_VEL
LIN {X 0,Y 107.748,Z 274.808,A -85,B 0,C 180,E1 -26219.785,E2 -26219.785} C_VEL
LIN {X 0,Y 106.376,Z 281.822,A -85,B 0,C 180,E1 -26224.164,E2 -26224.164} C_VEL
LIN {X 0,Y 105.361,Z 288.248,A -85,B 0,C 180,E1 -26229.364,E2 -26229.364} C_VEL
LIN {X 0,Y 104.994,Z 293.345,A -85,B 0,C 180,E1 -26234.831,E2 -26234.831} C_VEL
LIN {X 0,Y 105.145,Z 295.801,A -85,B 0,C 180,E1 -26238.06,E2 -26238.06} C_VEL
LIN {X 0,Y 106.034,Z 298.854,A -85,B 0,C 180,E1 -26243.383,E2 -26243.383} C_VEL
LIN {X 0,Y 107.764,Z 300.867,A -85,B 0,C 180,E1 -26248.556,E2 -26248.556} C_VEL
LIN {X 0,Y 110.311,Z 301.918,A -85,B 0,C 180,E1 -26253.518,E2 -26253.518} C_VEL
LIN {X 0,Y 113.579,Z 302.037,A -85,B 0,C 180,E1 -26258.21,E2 -26258.21} C_VEL
LIN {X 0,Y 117.733,Z 301.19,A -85,B 0,C 180,E1 -26262.766,E2 -26262.766} C_VEL
LIN {X 0,Y 122.621,Z 299.327,A -85,B 0,C 180,E1 -26266.994,E2 -26266.994} C_VEL
LIN {X 0,Y 128.121,Z 296.359,A -85,B 0,C 180,E1 -26270.886,E2 -26270.886} C_VEL
LIN {X 0,Y 133.289,Z 292.852,A -85,B 0,C 180,E1 -26273.949,E2 -26273.949} C_VEL
LIN {X 0,Y 134.723,Z 291.248,A -85,B 0,C 180,E1 -26275.503,E2 -26275.503} C_VEL
LIN {X 0,Y 136.59,Z 288.468,A -85,B 0,C 180,E1 -26278.528,E2 -26278.528} C_VEL
LIN {X 0,Y 137.603,Z 286.063,A -85,B 0,C 180,E1 -26281.466,E2 -26281.466} C_VEL
LIN {X 0,Y 138.332,Z 282.991,A -85,B 0,C 180,E1 -26285.834,E2 -26285.834} C_VEL
LIN {X 0,Y 138.346,Z 280.41,A -85,B 0,C 180,E1 -26291.727,E2 -26291.727} C_VEL
LIN {X 0,Y 137.816,Z 279.456,A -85,B 0,C 180,E1 -26297.819,E2 -26297.819} C_VEL
LIN {X 0,Y 137.808,Z 279.378,A -85,B 0,C 180,E1 -26300.918,E2 -26300.918} C_VEL
LIN {X 0,Y 137.695,Z 279.956,A -85,B 0,C 180,E1 -26304.102,E2 -26304.102} C_VEL
LIN {X 0,Y 137.625,Z 280.937,A -85,B 0,C 180,E1 -26307.364,E2 -26307.364} C_VEL
LIN {X 0,Y 137.807,Z 283.231,A -85,B 0,C 180,E1 -26312.38,E2 -26312.38} C_VEL
LIN {X 0,Y 137.383,Z 287.096,A -85,B 0,C 180,E1 -26317.873,E2 -26317.873} C_VEL
LIN {X 0,Y 136.929,Z 290.518,A -85,B 0,C 180,E1 -26321.857,E2 -26321.857} C_VEL
LIN {X 0,Y 136.188,Z 292.417,A -85,B 0,C 180,E1 -26323.742,E2 -26323.742} C_VEL
LIN {X 0,Y 133.157,Z 296.309,A -85,B 0,C 180,E1 -26326.675,E2 -26326.675} C_VEL
LIN {X 0,Y 129.908,Z 299.766,A -85,B 0,C 180,E1 -26329.52,E2 -26329.52} C_VEL
LIN {X 0,Y 126.301,Z 302.715,A -85,B 0,C 180,E1 -26332.26,E2 -26332.26} C_VEL
LIN {X 0,Y 122.312,Z 305.147,A -85,B 0,C 180,E1 -26334.929,E2 -26334.929} C_VEL
LIN {X 0,Y 118.769,Z 307.073,A -85,B 0,C 180,E1 -26337.822,E2 -26337.822} C_VEL
LIN {X 0,Y 115.505,Z 308.543,A -85,B 0,C 180,E1 -26340.872,E2 -26340.872} C_VEL
LIN {X 0,Y 112.666,Z 309.556,A -85,B 0,C 180,E1 -26344.11,E2 -26344.11} C_VEL
LIN {X 0,Y 110.306,Z 310.015,A -85,B 0,C 180,E1 -26347.526,E2 -26347.526} C_VEL
LIN {X 0,Y 108.457,Z 310.04,A -85,B 0,C 180,E1 -26351.096,E2 -26351.096} C_VEL
LIN {X 0,Y 107.064,Z 309.652,A -85,B 0,C 180,E1 -26354.778,E2 -26354.778} C_VEL
LIN {X 0,Y 106.143,Z 308.833,A -85,B 0,C 180,E1 -26358.543,E2 -26358.543} C_VEL
LIN {X 0,Y 105.683,Z 307.452,A -85,B 0,C 180,E1 -26362.358,E2 -26362.358} C_VEL
LIN {X 0,Y 105.782,Z 304.298,A -85,B 0,C 180,E1 -26368.417,E2 -26368.417} C_VEL
LIN {X 0,Y 105.831,Z 301.032,A -85,B 0,C 180,E1 -26372.746,E2 -26372.746} C_VEL
LIN {X 0,Y 105.965,Z 296.159,A -85,B 0,C 180,E1 -26377.623,E2 -26377.623} C_VEL
LIN {X 0,Y 106.625,Z 290.052,A -85,B 0,C 180,E1 -26382.37,E2 -26382.37} C_VEL
LIN {X 0,Y 107.578,Z 284.044,A -85,B 0,C 180,E1 -26386.121,E2 -26386.121} C_VEL
LIN {X 0,Y 108.957,Z 276.741,A -85,B 0,C 180,E1 -26389.795,E2 -26389.795} C_VEL
LIN {X 0,Y 109.086,Z 267.549,A -85,B 0,C 180,E1 -26393.547,E2 -26393.547} C_VEL
LIN {X 0,Y 109.011,Z 257.12,A -85,B 0,C 180,E1 -26396.828,E2 -26396.828} C_VEL
LIN {X 0,Y 108.884,Z 248.627,A -85,B 0,C 180,E1 -26398.954,E2 -26398.954} C_VEL
LIN {X 0,Y 108.528,Z 238.912,A -85,B 0,C 180,E1 -26400.865,E2 -26400.865} C_VEL
LIN {X 0,Y 108.396,Z 233.5,A -85,B 0,C 180,E1 -26401.806,E2 -26401.806} C_VEL
LIN {X 0,Y 108.962,Z 231.407,A -85,B 0,C 180,E1 -26405.486,E2 -26405.486} C_VEL
LIN {X 0,Y 108.234,Z 227.816,A -85,B 0,C 180,E1 -26412.414,E2 -26412.414} C_VEL
LIN {X 0,Y 107.724,Z 227.879,A -85,B 0,C 180,E1 -26421.528,E2 -26421.528} C_VEL
LIN {X 0,Y 107.805,Z 227.869,A -85,B 0,C 180,E1 -26428.561,E2 -26428.561} C_VEL
LIN {X 0,Y 107.915,Z 227.855,A -85,B 0,C 180,E1 -26436.996,E2 -26436.996} C_VEL
LIN {X 0,Y 108.034,Z 227.84,A -85,B 0,C 180,E1 -26444.914,E2 -26444.914} C_VEL
LIN {X 0,Y 108.257,Z 227.808,A -85,B 0,C 180,E1 -26448.766,E2 -26448.766} C_VEL
LIN {X 0,Y 108.449,Z 227.786,A -85,B 0,C 180,E1 -26456.281,E2 -26456.281} C_VEL
LIN {X 0,Y 108.945,Z 227.724,A -85,B 0,C 180,E1 -26459.997,E2 -26459.997} C_VEL
LIN {X 0,Y 108.302,Z 227.801,A -85,B 0,C 180,E1 -26467.454,E2 -26467.454} C_VEL
LIN {X 0,Y 108.14,Z 227.825,A -85,B 0,C 180,E1 -26472.874,E2 -26472.874} C_VEL
LIN {X 0,Y 107.884,Z 227.859,A -85,B 0,C 180,E1 -26479.006,E2 -26479.006} C_VEL
LIN {X 0,Y 107.856,Z 227.856,A -85,B 0,C 180,E1 -26484.18,E2 -26484.18} C_VEL
LIN {X 0,Y 107.793,Z 227.863,A -85,B 0,C 180,E1 -26492.048,E2 -26492.048} C_VEL
LIN {X 0,Y 107.705,Z 227.877,A -85,B 0,C 180,E1 -26498.46,E2 -26498.46} C_VEL
LIN {X 0,Y 107.67,Z 227.885,A -85,B 0,C 180,E1 -26503.938,E2 -26503.938} C_VEL
LIN {X 0,Y 107.438,Z 227.929,A -85,B 0,C 180,E1 -26506.022,E2 -26506.022} C_VEL
LIN {X 0,Y 106.691,Z 228.034,A -85,B 0,C 180,E1 -26508.087,E2 -26508.087} C_VEL
LIN {X 0,Y 104.345,Z 228.337,A -85,B 0,C 180,E1 -26512.203,E2 -26512.203} C_VEL
LIN {X 0,Y 101.015,Z 228.729,A -85,B 0,C 180,E1 -26518.754,E2 -26518.754} C_VEL
LIN {X 0,Y 100.645,Z 228.758,A -85,B 0,C 180,E1 -26521.049,E2 -26521.049} C_VEL
LIN {X 0,Y 100.781,Z 228.737,A -85,B 0,C 180,E1 -26525.265,E2 -26525.265} C_VEL
LIN {X 0,Y 100.811,Z 228.74,A -85,B 0,C 180,E1 -26529.599,E2 -26529.599} C_VEL
LIN {X 0,Y 101.182,Z 228.693,A -85,B 0,C 180,E1 -26537.972,E2 -26537.972} C_VEL
LIN {X 0,Y 101.261,Z 228.676,A -85,B 0,C 180,E1 -26542.02,E2 -26542.02} C_VEL
LIN {X 0,Y 101.859,Z 228.602,A -85,B 0,C 180,E1 -26549.999,E2 -26549.999} C_VEL
LIN {X 0,Y 101.133,Z 228.694,A -85,B 0,C 180,E1 -26557.988,E2 -26557.988} C_VEL
LIN {X 0,Y 100.562,Z 228.771,A -85,B 0,C 180,E1 -26563.45,E2 -26563.45} C_VEL
LIN {X 0,Y 101.985,Z 237.726,A -85,B 0,C 180,E1 -26565.488,E2 -26565.488} C_VEL
LIN {X 0,Y 102.965,Z 246.565,A -85,B 0,C 180,E1 -26567.887,E2 -26567.887} C_VEL
LIN {X 0,Y 103.706,Z 255.54,A -85,B 0,C 180,E1 -26570.841,E2 -26570.841} C_VEL
LIN {X 0,Y 103.82,Z 259.664,A -85,B 0,C 180,E1 -26572.381,E2 -26572.381} C_VEL
LIN {X 0,Y 102.015,Z 268.143,A -85,B 0,C 180,E1 -26575.993,E2 -26575.993} C_VEL
LIN {X 0,Y 100.481,Z 275.546,A -85,B 0,C 180,E1 -26579.977,E2 -26579.977} C_VEL
LIN {X 0,Y 98.969,Z 283.476,A -85,B 0,C 180,E1 -26585.445,E2 -26585.445} C_VEL
LIN {X 0,Y 98.174,Z 288.672,A -85,B 0,C 180,E1 -26590.111,E2 -26590.111} C_VEL
LIN {X 0,Y 97.947,Z 293.646,A -85,B 0,C 180,E1 -26595.85,E2 -26595.85} C_VEL
LIN {X 0,Y 98.524,Z 297.466,A -85,B 0,C 180,E1 -26601.688,E2 -26601.688} C_VEL
LIN {X 0,Y 100.06,Z 300.195,A -85,B 0,C 180,E1 -26607.441,E2 -26607.441} C_VEL
LIN {X 0,Y 102.562,Z 301.881,A -85,B 0,C 180,E1 -26612.975,E2 -26612.975} C_VEL
LIN {X 0,Y 105.956,Z 302.526,A -85,B 0,C 180,E1 -26618.218,E2 -26618.218} C_VEL
LIN {X 0,Y 110.175,Z 302.132,A -85,B 0,C 180,E1 -26623.104,E2 -26623.104} C_VEL
LIN {X 0,Y 115.134,Z 300.739,A -85,B 0,C 180,E1 -26627.597,E2 -26627.597} C_VEL
LIN {X 0,Y 120.744,Z 298.319,A -85,B 0,C 180,E1 -26631.686,E2 -26631.686} C_VEL
LIN {X 0,Y 125.447,Z 295.721,A -85,B 0,C 180,E1 -26634.556,E2 -26634.556} C_VEL
LIN {X 0,Y 126.917,Z 294.807,A -85,B 0,C 180,E1 -26635.372,E2 -26635.372} C_VEL
LIN {X 0,Y 128.741,Z 293.411,A -85,B 0,C 180,E1 -26636.873,E2 -26636.873} C_VEL
LIN {X 0,Y 130.72,Z 290.914,A -85,B 0,C 180,E1 -26640.003,E2 -26640.003} C_VEL
LIN {X 0,Y 131.806,Z 288.856,A -85,B 0,C 180,E1 -26643.059,E2 -26643.059} C_VEL
LIN {X 0,Y 132.482,Z 287.056,A -85,B 0,C 180,E1 -26646.093,E2 -26646.093} C_VEL
LIN {X 0,Y 132.724,Z 284.771,A -85,B 0,C 180,E1 -26652.231,E2 -26652.231} C_VEL
LIN {X 0,Y 132.422,Z 284.077,A -85,B 0,C 180,E1 -26658.571,E2 -26658.571} C_VEL
LIN {X 0,Y 132.418,Z 284.197,A -85,B 0,C 180,E1 -26661.812,E2 -26661.812} C_VEL
LIN {X 0,Y 132.214,Z 284.969,A -85,B 0,C 180,E1 -26665.358,E2 -26665.358} C_VEL
LIN {X 0,Y 132.125,Z 286.007,A -85,B 0,C 180,E1 -26668.605,E2 -26668.605} C_VEL
LIN {X 0,Y 132.119,Z 287.536,A -85,B 0,C 180,E1 -26672.14,E2 -26672.14} C_VEL
LIN {X 0,Y 131.539,Z 290.409,A -85,B 0,C 180,E1 -26676.733,E2 -26676.733} C_VEL
LIN {X 0,Y 130.726,Z 293.678,A -85,B 0,C 180,E1 -26681.179,E2 -26681.179} C_VEL
LIN {X 0,Y 129.674,Z 295.43,A -85,B 0,C 180,E1 -26682.974,E2 -26682.974} C_VEL
LIN {X 0,Y 125.054,Z 299.95,A -85,B 0,C 180,E1 -26686.94,E2 -26686.94} C_VEL
LIN {X 0,Y 120.78,Z 303.182,A -85,B 0,C 180,E1 -26690.203,E2 -26690.203} C_VEL
LIN {X 0,Y 116.578,Z 305.48,A -85,B 0,C 180,E1 -26692.926,E2 -26692.926} C_VEL
LIN {X 0,Y 112.825,Z 307.204,A -85,B 0,C 180,E1 -26695.902,E2 -26695.902} C_VEL
LIN {X 0,Y 109.362,Z 308.486,A -85,B 0,C 180,E1 -26699.063,E2 -26699.063} C_VEL
LIN {X 0,Y 106.328,Z 309.338,A -85,B 0,C 180,E1 -26702.441,E2 -26702.441} C_VEL
LIN {X 0,Y 103.764,Z 309.75,A -85,B 0,C 180,E1 -26706.023,E2 -26706.023} C_VEL
LIN {X 0,Y 101.762,Z 309.614,A -85,B 0,C 180,E1 -26709.8,E2 -26709.8} C_VEL
LIN {X 0,Y 100.237,Z 309.054,A -85,B 0,C 180,E1 -26713.713,E2 -26713.713} C_VEL
LIN {X 0,Y 99.218,Z 308.083,A -85,B 0,C 180,E1 -26717.732,E2 -26717.732} C_VEL
LIN {X 0,Y 98.698,Z 306.65,A -85,B 0,C 180,E1 -26721.813,E2 -26721.813} C_VEL
LIN {X 0,Y 98.781,Z 303.198,A -85,B 0,C 180,E1 -26728.27,E2 -26728.27} C_VEL
LIN {X 0,Y 98.799,Z 299.927,A -85,B 0,C 180,E1 -26732.693,E2 -26732.693} C_VEL
LIN {X 0,Y 98.995,Z 294.594,A -85,B 0,C 180,E1 -26738.164,E2 -26738.164} C_VEL
LIN {X 0,Y 99.543,Z 289.636,A -85,B 0,C 180,E1 -26742.229,E2 -26742.229} C_VEL
LIN {X 0,Y 100.496,Z 283.637,A -85,B 0,C 180,E1 -26746.245,E2 -26746.245} C_VEL
LIN {X 0,Y 101.895,Z 276.346,A -85,B 0,C 180,E1 -26750.174,E2 -26750.174} C_VEL
LIN {X 0,Y 102.03,Z 266.518,A -85,B 0,C 180,E1 -26754.412,E2 -26754.412} C_VEL
LIN {X 0,Y 102.012,Z 256.439,A -85,B 0,C 180,E1 -26757.745,E2 -26757.745} C_VEL
LIN {X 0,Y 101.884,Z 247.885,A -85,B 0,C 180,E1 -26760.008,E2 -26760.008} C_VEL
LIN {X 0,Y 101.66,Z 237.62,A -85,B 0,C 180,E1 -26762.105,E2 -26762.105} C_VEL
LIN {X 0,Y 101.523,Z 233.305,A -85,B 0,C 180,E1 -26762.888,E2 -26762.888} C_VEL
LIN {X 0,Y 101.792,Z 231.692,A -85,B 0,C 180,E1 -26765.956,E2 -26765.956} C_VEL
LIN {X 0,Y 101.201,Z 228.692,A -85,B 0,C 180,E1 -26771.98,E2 -26771.98} C_VEL
LIN {X 0,Y 100.669,Z 228.757,A -85,B 0,C 180,E1 -26781.07,E2 -26781.07} C_VEL
LIN {X 0,Y 100.7,Z 228.752,A -85,B 0,C 180,E1 -26786.878,E2 -26786.878} C_VEL
LIN {X 0,Y 100.79,Z 228.74,A -85,B 0,C 180,E1 -26795.265,E2 -26795.265} C_VEL
LIN {X 0,Y 100.82,Z 228.736,A -85,B 0,C 180,E1 -26799.598,E2 -26799.598} C_VEL
LIN {X 0,Y 101.106,Z 228.703,A -85,B 0,C 180,E1 -26806.699,E2 -26806.699} C_VEL
LIN {X 0,Y 101.246,Z 228.684,A -85,B 0,C 180,E1 -26812.016,E2 -26812.016} C_VEL
LIN {X 0,Y 101.869,Z 228.606,A -85,B 0,C 180,E1 -26819.997,E2 -26819.997} C_VEL
LIN {X 0,Y 101.237,Z 228.683,A -85,B 0,C 180,E1 -26827.977,E2 -26827.977} C_VEL
LIN {X 0,Y 101.055,Z 228.706,A -85,B 0,C 180,E1 -26833.179,E2 -26833.179} C_VEL
LIN {X 0,Y 100.802,Z 228.741,A -85,B 0,C 180,E1 -26840.398,E2 -26840.398} C_VEL
LIN {X 0,Y 100.774,Z 228.741,A -85,B 0,C 180,E1 -26844.955,E2 -26844.955} C_VEL
LIN {X 0,Y 100.698,Z 228.75,A -85,B 0,C 180,E1 -26853.12,E2 -26853.12} C_VEL
LIN {X 0,Y 100.652,Z 228.753,A -85,B 0,C 180,E1 -26859.817,E2 -26859.817} C_VEL
LIN {X 0,Y 100.647,Z 228.76,A -85,B 0,C 180,E1 -26865.709,E2 -26865.709} C_VEL
LIN {X 0,Y 100.623,Z 228.762,A -85,B 0,C 180,E1 -26871.052,E2 -26871.052} C_VEL
LIN {X 0,Y 100.686,Z 228.748,A -85,B 0,C 180,E1 -26876.882,E2 -26876.882} C_VEL
LIN {X 0,Y 100.645,Z 228.758,A -85,B 0,C 180,E1 -26881.049,E2 -26881.049} C_VEL
LIN {X 0,Y 99.945,Z 228.842,A -85,B 0,C 180,E1 -26884.394,E2 -26884.394} C_VEL
LIN {X 0,Y 98.437,Z 229.035,A -85,B 0,C 180,E1 -26887.714,E2 -26887.714} C_VEL
LIN {X 0,Y 94.299,Z 229.551,A -85,B 0,C 180,E1 -26896.987,E2 -26896.987} C_VEL
LIN {X 0,Y 94.077,Z 229.566,A -85,B 0,C 180,E1 -26899.439,E2 -26899.439} C_VEL
LIN {X 0,Y 94.298,Z 229.551,A -85,B 0,C 180,E1 -26905.725,E2 -26905.725} C_VEL
LIN {X 0,Y 94.783,Z 229.483,A -85,B 0,C 180,E1 -26909.999,E2 -26909.999} C_VEL
LIN {X 0,Y 94,Z 229.581,A -85,B 0,C 180,E1 -26918.599,E2 -26918.599} C_VEL
LIN {X 0,Y 93.693,Z 229.627,A -85,B 0,C 180,E1 -26922.276,E2 -26922.276} C_VEL
LIN {X 0,Y 95.062,Z 238.36,A -85,B 0,C 180,E1 -26924.448,E2 -26924.448} C_VEL
LIN {X 0,Y 96.008,Z 247.112,A -85,B 0,C 180,E1 -26927.025,E2 -26927.025} C_VEL
LIN {X 0,Y 96.695,Z 256.027,A -85,B 0,C 180,E1 -26930.195,E2 -26930.195} C_VEL
LIN {X 0,Y 96.719,Z 260.172,A -85,B 0,C 180,E1 -26931.863,E2 -26931.863} C_VEL
LIN {X 0,Y 95.121,Z 267.467,A -85,B 0,C 180,E1 -26935.14,E2 -26935.14} C_VEL
LIN {X 0,Y 93.551,Z 274.741,A -85,B 0,C 180,E1 -26939.226,E2 -26939.226} C_VEL
LIN {X 0,Y 92.15,Z 281.611,A -85,B 0,C 180,E1 -26944.099,E2 -26944.099} C_VEL
LIN {X 0,Y 91.143,Z 287.698,A -85,B 0,C 180,E1 -26949.554,E2 -26949.554} C_VEL
LIN {X 0,Y 90.862,Z 293.102,A -85,B 0,C 180,E1 -26955.888,E2 -26955.888} C_VEL
LIN {X 0,Y 91.46,Z 297.073,A -85,B 0,C 180,E1 -26962.072,E2 -26962.072} C_VEL
LIN {X 0,Y 93.035,Z 299.945,A -85,B 0,C 180,E1 -26968.081,E2 -26968.081} C_VEL
LIN {X 0,Y 95.597,Z 301.82,A -85,B 0,C 180,E1 -26973.83,E2 -26973.83} C_VEL
LIN {X 0,Y 99.04,Z 302.738,A -85,B 0,C 180,E1 -26979.222,E2 -26979.222} C_VEL
LIN {X 0,Y 103.277,Z 302.737,A -85,B 0,C 180,E1 -26984.208,E2 -26984.208} C_VEL
LIN {X 0,Y 108.241,Z 301.816,A -85,B 0,C 180,E1 -26988.771,E2 -26988.771} C_VEL
LIN {X 0,Y 113.873,Z 299.936,A -85,B 0,C 180,E1 -26992.913,E2 -26992.913} C_VEL
LIN {X 0,Y 120.075,Z 297.002,A -85,B 0,C 180,E1 -26996.647,E2 -26996.647} C_VEL
LIN {X 0,Y 122.689,Z 295.36,A -85,B 0,C 180,E1 -26998.362,E2 -26998.362} C_VEL
LIN {X 0,Y 123.922,Z 294.315,A -85,B 0,C 180,E1 -27000.003,E2 -27000.003} C_VEL
LIN {X 0,Y 125.45,Z 292.332,A -85,B 0,C 180,E1 -27003.214,E2 -27003.214} C_VEL
LIN {X 0,Y 126.41,Z 290.791,A -85,B 0,C 180,E1 -27006.387,E2 -27006.387} C_VEL
LIN {X 0,Y 126.673,Z 289.662,A -85,B 0,C 180,E1 -27009.584,E2 -27009.584} C_VEL
LIN {X 0,Y 126.872,Z 288.779,A -85,B 0,C 180,E1 -27012.804,E2 -27012.804} C_VEL
LIN {X 0,Y 126.727,Z 288.382,A -85,B 0,C 180,E1 -27019.477,E2 -27019.477} C_VEL
LIN {X 0,Y 126.642,Z 288.723,A -85,B 0,C 180,E1 -27022.862,E2 -27022.862} C_VEL
LIN {X 0,Y 126.354,Z 289.726,A -85,B 0,C 180,E1 -27027.135,E2 -27027.135} C_VEL
LIN {X 0,Y 126.262,Z 290.7,A -85,B 0,C 180,E1 -27030.066,E2 -27030.066} C_VEL
LIN {X 0,Y 125.813,Z 292.546,A -85,B 0,C 180,E1 -27033.962,E2 -27033.962} C_VEL
LIN {X 0,Y 124.952,Z 295.099,A -85,B 0,C 180,E1 -27038.224,E2 -27038.224} C_VEL
LIN {X 0,Y 124.387,Z 296.474,A -85,B 0,C 180,E1 -27040.374,E2 -27040.374} C_VEL
LIN {X 0,Y 123.013,Z 298.04,A -85,B 0,C 180,E1 -27042.037,E2 -27042.037} C_VEL
LIN {X 0,Y 117.423,Z 302.398,A -85,B 0,C 180,E1 -27046.505,E2 -27046.505} C_VEL
LIN {X 0,Y 113.172,Z 304.709,A -85,B 0,C 180,E1 -27049.304,E2 -27049.304} C_VEL
LIN {X 0,Y 107.025,Z 307.356,A -85,B 0,C 180,E1 -27053.773,E2 -27053.773} C_VEL
LIN {X 0,Y 103.344,Z 308.44,A -85,B 0,C 180,E1 -27057.041,E2 -27057.041} C_VEL
LIN {X 0,Y 100.095,Z 309.098,A -85,B 0,C 180,E1 -27060.562,E2 -27060.562} C_VEL
LIN {X 0,Y 97.309,Z 309.35,A -85,B 0,C 180,E1 -27064.321,E2 -27064.321} C_VEL
LIN {X 0,Y 95.132,Z 309.171,A -85,B 0,C 180,E1 -27068.323,E2 -27068.323} C_VEL
LIN {X 0,Y 93.455,Z 308.443,A -85,B 0,C 180,E1 -27072.495,E2 -27072.495} C_VEL
LIN {X 0,Y 92.321,Z 307.284,A -85,B 0,C 180,E1 -27076.799,E2 -27076.799} C_VEL
LIN {X 0,Y 91.696,Z 303.878,A -85,B 0,C 180,E1 -27085.159,E2 -27085.159} C_VEL
LIN {X 0,Y 91.867,Z 300.891,A -85,B 0,C 180,E1 -27090.001,E2 -27090.001} C_VEL
LIN {X 0,Y 91.825,Z 295.513,A -85,B 0,C 180,E1 -27096.373,E2 -27096.373} C_VEL
LIN {X 0,Y 92.271,Z 290.556,A -85,B 0,C 180,E1 -27100.978,E2 -27100.978} C_VEL
LIN {X 0,Y 93.149,Z 284.82,A -85,B 0,C 180,E1 -27105.313,E2 -27105.313} C_VEL
LIN {X 0,Y 94.468,Z 277.824,A -85,B 0,C 180,E1 -27109.56,E2 -27109.56} C_VEL
LIN {X 0,Y 94.865,Z 273.682,A -85,B 0,C 180,E1 -27111.742,E2 -27111.742} C_VEL
LIN {X 0,Y 94.979,Z 264.343,A -85,B 0,C 180,E1 -27115.769,E2 -27115.769} C_VEL
LIN {X 0,Y 95.032,Z 254.858,A -85,B 0,C 180,E1 -27119.04,E2 -27119.04} C_VEL
LIN {X 0,Y 94.908,Z 244.554,A -85,B 0,C 180,E1 -27121.845,E2 -27121.845} C_VEL
LIN {X 0,Y 94.597,Z 233.047,A -85,B 0,C 180,E1 -27124.185,E2 -27124.185} C_VEL
LIN {X 0,Y 94.623,Z 231.947,A -85,B 0,C 180,E1 -27126.456,E2 -27126.456} C_VEL
LIN {X 0,Y 94.19,Z 229.566,A -85,B 0,C 180,E1 -27131.737,E2 -27131.737} C_VEL
LIN {X 0,Y 93.647,Z 229.63,A -85,B 0,C 180,E1 -27138.633,E2 -27138.633} C_VEL
LIN {X 0,Y 93.601,Z 229.631,A -85,B 0,C 180,E1 -27145.685,E2 -27145.685} C_VEL
LIN {X 0,Y 93.673,Z 229.623,A -85,B 0,C 180,E1 -27154.203,E2 -27154.203} C_VEL
LIN {X 0,Y 93.697,Z 229.626,A -85,B 0,C 180,E1 -27157.97,E2 -27157.97} C_VEL
LIN {X 0,Y 94.026,Z 229.585,A -85,B 0,C 180,E1 -27166.339,E2 -27166.339} C_VEL
LIN {X 0,Y 94.179,Z 229.561,A -85,B 0,C 180,E1 -27171.413,E2 -27171.413} C_VEL
LIN {X 0,Y 94.794,Z 229.486,A -85,B 0,C 180,E1 -27179.996,E2 -27179.996} C_VEL
LIN {X 0,Y 94.166,Z 229.564,A -85,B 0,C 180,E1 -27188.581,E2 -27188.581} C_VEL
LIN {X 0,Y 93.964,Z 229.589,A -85,B 0,C 180,E1 -27193.507,E2 -27193.507} C_VEL
LIN {X 0,Y 93.684,Z 229.623,A -85,B 0,C 180,E1 -27202.026,E2 -27202.026} C_VEL
LIN {X 0,Y 93.623,Z 229.636,A -85,B 0,C 180,E1 -27206.765,E2 -27206.765} C_VEL
LIN {X 0,Y 93.597,Z 229.637,A -85,B 0,C 180,E1 -27214.311,E2 -27214.311} C_VEL
LIN {X 0,Y 93.536,Z 229.645,A -85,B 0,C 180,E1 -27222.544,E2 -27222.544} C_VEL
LIN {X 0,Y 93.532,Z 229.639,A -85,B 0,C 180,E1 -27228.706,E2 -27228.706} C_VEL
LIN {X 0,Y 93.583,Z 229.634,A -85,B 0,C 180,E1 -27235.692,E2 -27235.692} C_VEL
LIN {X 0,Y 93.664,Z 229.625,A -85,B 0,C 180,E1 -27244.203,E2 -27244.203} C_VEL
LIN {X 0,Y 93.688,Z 229.627,A -85,B 0,C 180,E1 -27247.97,E2 -27247.97} C_VEL
LIN {X 0,Y 94.086,Z 229.578,A -85,B 0,C 180,E1 -27257.05,E2 -27257.05} C_VEL
LIN {X 0,Y 94.077,Z 229.566,A -85,B 0,C 180,E1 -27259.439,E2 -27259.439} C_VEL
LIN {X 0,Y 93.81,Z 229.604,A -85,B 0,C 180,E1 -27261.831,E2 -27261.831} C_VEL
LIN {X 0,Y 92.478,Z 229.778,A -85,B 0,C 180,E1 -27265.384,E2 -27265.384} C_VEL
LIN {X 0,Y 89.226,Z 230.18,A -85,B 0,C 180,E1 -27271.398,E2 -27271.398} C_VEL
LIN {X 0,Y 87.199,Z 230.432,A -85,B 0,C 180,E1 -27276.548,E2 -27276.548} C_VEL
LIN {X 0,Y 86.878,Z 230.468,A -85,B 0,C 180,E1 -27279.227,E2 -27279.227} C_VEL
LIN {X 0,Y 86.767,Z 230.642,A -85,B 0,C 180,E1 -27281.073,E2 -27281.073} C_VEL
LIN {X 0,Y 87.986,Z 237.237,A -85,B 0,C 180,E1 -27282.827,E2 -27282.827} C_VEL
LIN {X 0,Y 89.04,Z 247.435,A -85,B 0,C 180,E1 -27286.036,E2 -27286.036} C_VEL
LIN {X 0,Y 89.696,Z 256.599,A -85,B 0,C 180,E1 -27289.548,E2 -27289.548} C_VEL
LIN {X 0,Y 89.738,Z 260.083,A -85,B 0,C 180,E1 -27291.053,E2 -27291.053} C_VEL
LIN {X 0,Y 87.978,Z 267.776,A -85,B 0,C 180,E1 -27294.779,E2 -27294.779} C_VEL
LIN {X 0,Y 86.319,Z 275.089,A -85,B 0,C 180,E1 -27299.242,E2 -27299.242} C_VEL
LIN {X 0,Y 84.989,Z 281.595,A -85,B 0,C 180,E1 -27304.223,E2 -27304.223} C_VEL
LIN {X 0,Y 83.943,Z 288.643,A -85,B 0,C 180,E1 -27311.111,E2 -27311.111} C_VEL
LIN {X 0,Y 83.896,Z 293.826,A -85,B 0,C 180,E1 -27317.926,E2 -27317.926} C_VEL
LIN {X 0,Y 84.82,Z 297.684,A -85,B 0,C 180,E1 -27324.555,E2 -27324.555} C_VEL
LIN {X 0,Y 86.837,Z 300.465,A -85,B 0,C 180,E1 -27330.953,E2 -27330.953} C_VEL
LIN {X 0,Y 90.734,Z 302.615,A -85,B 0,C 180,E1 -27338.354,E2 -27338.354} C_VEL
LIN {X 0,Y 95.051,Z 303.261,A -85,B 0,C 180,E1 -27343.986,E2 -27343.986} C_VEL
LIN {X 0,Y 100.206,Z 302.892,A -85,B 0,C 180,E1 -27349.077,E2 -27349.077} C_VEL
LIN {X 0,Y 106.075,Z 301.541,A -85,B 0,C 180,E1 -27353.624,E2 -27353.624} C_VEL
LIN {X 0,Y 112.542,Z 299.194,A -85,B 0,C 180,E1 -27357.651,E2 -27357.651} C_VEL
LIN {X 0,Y 116.601,Z 297.32,A -85,B 0,C 180,E1 -27360.003,E2 -27360.003} C_VEL
LIN {X 0,Y 118.797,Z 295.488,A -85,B 0,C 180,E1 -27363.394,E2 -27363.394} C_VEL
LIN {X 0,Y 120.074,Z 294.076,A -85,B 0,C 180,E1 -27366.725,E2 -27366.725} C_VEL
LIN {X 0,Y 120.529,Z 293.1,A -85,B 0,C 180,E1 -27370.077,E2 -27370.077} C_VEL
LIN {X 0,Y 120.784,Z 292.47,A -85,B 0,C 180,E1 -27373.462,E2 -27373.462} C_VEL
LIN {X 0,Y 120.716,Z 292.312,A -85,B 0,C 180,E1 -27376.926,E2 -27376.926} C_VEL
LIN {X 0,Y 120.688,Z 292.439,A -85,B 0,C 180,E1 -27381.296,E2 -27381.296} C_VEL
LIN {X 0,Y 120.538,Z 292.87,A -85,B 0,C 180,E1 -27384.091,E2 -27384.091} C_VEL
LIN {X 0,Y 120.209,Z 293.98,A -85,B 0,C 180,E1 -27388.721,E2 -27388.721} C_VEL
LIN {X 0,Y 119.849,Z 295.102,A -85,B 0,C 180,E1 -27391.857,E2 -27391.857} C_VEL
LIN {X 0,Y 118.933,Z 297.188,A -85,B 0,C 180,E1 -27396.226,E2 -27396.226} C_VEL
LIN {X 0,Y 118.039,Z 298.885,A -85,B 0,C 180,E1 -27399.285,E2 -27399.285} C_VEL
LIN {X 0,Y 116.302,Z 300.24,A -85,B 0,C 180,E1 -27400.944,E2 -27400.944} C_VEL
LIN {X 0,Y 112.232,Z 302.881,A -85,B 0,C 180,E1 -27404.06,E2 -27404.06} C_VEL
LIN {X 0,Y 110.211,Z 303.945,A -85,B 0,C 180,E1 -27405.457,E2 -27405.457} C_VEL
LIN {X 0,Y 105.603,Z 305.88,A -85,B 0,C 180,E1 -27408.279,E2 -27408.279} C_VEL
LIN {X 0,Y 101.376,Z 307.368,A -85,B 0,C 180,E1 -27411.397,E2 -27411.397} C_VEL
LIN {X 0,Y 97.472,Z 308.391,A -85,B 0,C 180,E1 -27414.774,E2 -27414.774} C_VEL
LIN {X 0,Y 93.987,Z 308.865,A -85,B 0,C 180,E1 -27418.438,E2 -27418.438} C_VEL
LIN {X 0,Y 90.956,Z 308.918,A -85,B 0,C 180,E1 -27422.381,E2 -27422.381} C_VEL
LIN {X 0,Y 88.578,Z 308.588,A -85,B 0,C 180,E1 -27426.628,E2 -27426.628} C_VEL
LIN {X 0,Y 86.727,Z 307.817,A -85,B 0,C 180,E1 -27431.087,E2 -27431.087} C_VEL
LIN {X 0,Y 85.458,Z 306.488,A -85,B 0,C 180,E1 -27435.718,E2 -27435.718} C_VEL
LIN {X 0,Y 84.702,Z 302.746,A -85,B 0,C 180,E1 -27444.708,E2 -27444.708} C_VEL
LIN {X 0,Y 84.874,Z 299.595,A -85,B 0,C 180,E1 -27450.001,E2 -27450.001} C_VEL
LIN {X 0,Y 84.779,Z 294.915,A -85,B 0,C 180,E1 -27455.828,E2 -27455.828} C_VEL
LIN {X 0,Y 85.202,Z 290.079,A -85,B 0,C 180,E1 -27460.697,E2 -27460.697} C_VEL
LIN {X 0,Y 86.061,Z 284.342,A -85,B 0,C 180,E1 -27465.392,E2 -27465.392} C_VEL
LIN {X 0,Y 87.602,Z 276.337,A -85,B 0,C 180,E1 -27470.549,E2 -27470.549} C_VEL
LIN {X 0,Y 87.864,Z 270.626,A -85,B 0,C 180,E1 -27473.575,E2 -27473.575} C_VEL
LIN {X 0,Y 87.965,Z 262.15,A -85,B 0,C 180,E1 -27477.349,E2 -27477.349} C_VEL
LIN {X 0,Y 88.077,Z 253.165,A -85,B 0,C 180,E1 -27480.578,E2 -27480.578} C_VEL
LIN {X 0,Y 88.002,Z 240.901,A -85,B 0,C 180,E1 -27483.904,E2 -27483.904} C_VEL
LIN {X 0,Y 87.779,Z 234.448,A -85,B 0,C 180,E1 -27485.275,E2 -27485.275} C_VEL
LIN {X 0,Y 87.571,Z 232.758,A -85,B 0,C 180,E1 -27485.742,E2 -27485.742} C_VEL
LIN {X 0,Y 87.159,Z 230.442,A -85,B 0,C 180,E1 -27491.399,E2 -27491.399} C_VEL
LIN {X 0,Y 86.54,Z 230.517,A -85,B 0,C 180,E1 -27499.477,E2 -27499.477} C_VEL
LIN {X 0,Y 86.547,Z 230.509,A -85,B 0,C 180,E1 -27505.355,E2 -27505.355} C_VEL
LIN {X 0,Y 86.588,Z 230.504,A -85,B 0,C 180,E1 -27513.233,E2 -27513.233} C_VEL
LIN {X 0,Y 86.649,Z 230.497,A -85,B 0,C 180,E1 -27521.065,E2 -27521.065} C_VEL
LIN {X 0,Y 86.934,Z 230.469,A -85,B 0,C 180,E1 -27525.96,E2 -27525.96} C_VEL
LIN {X 0,Y 87.088,Z 230.443,A -85,B 0,C 180,E1 -27530.708,E2 -27530.708} C_VEL
LIN {X 0,Y 87.72,Z 230.367,A -85,B 0,C 180,E1 -27539.996,E2 -27539.996} C_VEL
LIN {X 0,Y 87.068,Z 230.451,A -85,B 0,C 180,E1 -27549.286,E2 -27549.286} C_VEL
LIN {X 0,Y 86.861,Z 230.472,A -85,B 0,C 180,E1 -27554.044,E2 -27554.044} C_VEL
LIN {X 0,Y 86.619,Z 230.508,A -85,B 0,C 180,E1 -27558.934,E2 -27558.934} C_VEL
LIN {X 0,Y 86.584,Z 230.513,A -85,B 0,C 180,E1 -27566.762,E2 -27566.762} C_VEL
LIN {X 0,Y 86.515,Z 230.521,A -85,B 0,C 180,E1 -27575.673,E2 -27575.673} C_VEL
LIN {X 0,Y 86.478,Z 230.525,A -85,B 0,C 180,E1 -27582.992,E2 -27582.992} C_VEL
LIN {X 0,Y 86.453,Z 230.522,A -85,B 0,C 180,E1 -27589.432,E2 -27589.432} C_VEL
LIN {X 0,Y 86.526,Z 230.514,A -85,B 0,C 180,E1 -27595.348,E2 -27595.348} C_VEL
LIN {X 0,Y 86.579,Z 230.509,A -85,B 0,C 180,E1 -27603.232,E2 -27603.232} C_VEL
LIN {X 0,Y 86.657,Z 230.501,A -85,B 0,C 180,E1 -27611.07,E2 -27611.07} C_VEL
LIN {X 0,Y 86.964,Z 230.464,A -85,B 0,C 180,E1 -27615.968,E2 -27615.968} C_VEL
LIN {X 0,Y 87.102,Z 230.441,A -85,B 0,C 180,E1 -27620.712,E2 -27620.712} C_VEL
LIN {X 0,Y 87.707,Z 230.365,A -85,B 0,C 180,E1 -27629.999,E2 -27629.999} C_VEL
LIN {X 0,Y 86.878,Z 230.468,A -85,B 0,C 180,E1 -27639.227,E2 -27639.227} C_VEL
LIN {X 0,Y 86.871,Z 231.369,A -85,B 0,C 180,E1 -27640.536,E2 -27640.536} C_VEL
LIN {X 0,Y 86.797,Z 234.706,A -85,B 0,C 180,E1 -27641.957,E2 -27641.957} C_VEL
LIN {X 0,Y 86.394,Z 240.489,A -85,B 0,C 180,E1 -27643.407,E2 -27643.407} C_VEL
LIN {X 0,Y 84.941,Z 247.38,A -85,B 0,C 180,E1 -27645.301,E2 -27645.301} C_VEL
LIN {X 0,Y 83.202,Z 254.285,A -85,B 0,C 180,E1 -27647.506,E2 -27647.506} C_VEL
LIN {X 0,Y 82.758,Z 258.187,A -85,B 0,C 180,E1 -27649.284,E2 -27649.284} C_VEL
LIN {X 0,Y 82.549,Z 260.801,A -85,B 0,C 180,E1 -27650.541,E2 -27650.541} C_VEL
LIN {X 0,Y 80.799,Z 268.251,A -85,B 0,C 180,E1 -27654.479,E2 -27654.479} C_VEL
LIN {X 0,Y 79.254,Z 274.789,A -85,B 0,C 180,E1 -27658.776,E2 -27658.776} C_VEL
LIN {X 0,Y 77.898,Z 281.198,A -85,B 0,C 180,E1 -27664.02,E2 -27664.02} C_VEL
LIN {X 0,Y 76.976,Z 286.776,A -85,B 0,C 180,E1 -27669.724,E2 -27669.724} C_VEL
LIN {X 0,Y 76.765,Z 292.471,A -85,B 0,C 180,E1 -27677.088,E2 -27677.088} C_VEL
LIN {X 0,Y 77.66,Z 296.896,A -85,B 0,C 180,E1 -27684.534,E2 -27684.534} C_VEL
LIN {X 0,Y 80.873,Z 300.968,A -85,B 0,C 180,E1 -27694.251,E2 -27694.251} C_VEL
LIN {X 0,Y 84.462,Z 302.726,A -85,B 0,C 180,E1 -27700.564,E2 -27700.564} C_VEL
LIN {X 0,Y 89.003,Z 303.547,A -85,B 0,C 180,E1 -27706.301,E2 -27706.301} C_VEL
LIN {X 0,Y 94.373,Z 303.452,A -85,B 0,C 180,E1 -27711.438,E2 -27711.438} C_VEL
LIN {X 0,Y 100.453,Z 302.423,A -85,B 0,C 180,E1 -27715.992,E2 -27715.992} C_VEL
LIN {X 0,Y 107.182,Z 300.395,A -85,B 0,C 180,E1 -27720.003,E2 -27720.003} C_VEL
LIN {X 0,Y 110.44,Z 299.036,A -85,B 0,C 180,E1 -27721.826,E2 -27721.826} C_VEL
LIN {X 0,Y 111.831,Z 298.296,A -85,B 0,C 180,E1 -27723.606,E2 -27723.606} C_VEL
LIN {X 0,Y 113.555,Z 296.955,A -85,B 0,C 180,E1 -27727.113,E2 -27727.113} C_VEL
LIN {X 0,Y 114.193,Z 296.194,A -85,B 0,C 180,E1 -27730.643,E2 -27730.643} C_VEL
LIN {X 0,Y 114.479,Z 295.792,A -85,B 0,C 180,E1 -27734.218,E2 -27734.218} C_VEL
LIN {X 0,Y 114.452,Z 295.705,A -85,B 0,C 180,E1 -27737.883,E2 -27737.883} C_VEL
LIN {X 0,Y 114.342,Z 296.051,A -85,B 0,C 180,E1 -27742.785,E2 -27742.785} C_VEL
LIN {X 0,Y 114.106,Z 296.567,A -85,B 0,C 180,E1 -27745.543,E2 -27745.543} C_VEL
LIN {X 0,Y 113.65,Z 297.707,A -85,B 0,C 180,E1 -27750.033,E2 -27750.033} C_VEL
LIN {X 0,Y 112.905,Z 299.099,A -85,B 0,C 180,E1 -27754.075,E2 -27754.075} C_VEL
LIN {X 0,Y 111.545,Z 300.946,A -85,B 0,C 180,E1 -27758.041,E2 -27758.041} C_VEL
LIN {X 0,Y 108.83,Z 302.552,A -85,B 0,C 180,E1 -27760.228,E2 -27760.228} C_VEL
LIN {X 0,Y 105.24,Z 304.373,A -85,B 0,C 180,E1 -27762.729,E2 -27762.729} C_VEL
LIN {X 0,Y 100.419,Z 306.077,A -85,B 0,C 180,E1 -27765.584,E2 -27765.584} C_VEL
LIN {X 0,Y 95.922,Z 307.342,A -85,B 0,C 180,E1 -27768.746,E2 -27768.746} C_VEL
LIN {X 0,Y 91.774,Z 308.197,A -85,B 0,C 180,E1 -27772.221,E2 -27772.221} C_VEL
LIN {X 0,Y 88.029,Z 308.616,A -85,B 0,C 180,E1 -27776.024,E2 -27776.024} C_VEL
LIN {X 0,Y 84.725,Z 308.486,A -85,B 0,C 180,E1 -27780.153,E2 -27780.153} C_VEL
LIN {X 0,Y 80.064,Z 307.025,A -85,B 0,C 180,E1 -27789.445,E2 -27789.445} C_VEL
LIN {X 0,Y 78.635,Z 305.656,A -85,B 0,C 180,E1 -27794.448,E2 -27794.448} C_VEL
LIN {X 0,Y 77.695,Z 302.58,A -85,B 0,C 180,E1 -27802.205,E2 -27802.205} C_VEL
LIN {X 0,Y 77.78,Z 300.106,A -85,B 0,C 180,E1 -27807.014,E2 -27807.014} C_VEL
LIN {X 0,Y 77.801,Z 297.147,A -85,B 0,C 180,E1 -27811.473,E2 -27811.473} C_VEL
LIN {X 0,Y 78.003,Z 290.847,A -85,B 0,C 180,E1 -27819.072,E2 -27819.072} C_VEL
LIN {X 0,Y 78.993,Z 283.722,A -85,B 0,C 180,E1 -27825.481,E2 -27825.481} C_VEL
LIN {X 0,Y 80.401,Z 276.686,A -85,B 0,C 180,E1 -27830.467,E2 -27830.467} C_VEL
LIN {X 0,Y 80.796,Z 271.162,A -85,B 0,C 180,E1 -27833.723,E2 -27833.723} C_VEL
LIN {X 0,Y 80.941,Z 263.34,A -85,B 0,C 180,E1 -27837.601,E2 -27837.601} C_VEL
LIN {X 0,Y 81.126,Z 255.447,A -85,B 0,C 180,E1 -27840.819,E2 -27840.819} C_VEL
LIN {X 0,Y 81.194,Z 246.18,A -85,B 0,C 180,E1 -27843.865,E2 -27843.865} C_VEL
LIN {X 0,Y 80.945,Z 234.992,A -85,B 0,C 180,E1 -27846.711,E2 -27846.711} C_VEL
LIN {X 0,Y 80.356,Z 232.525,A -85,B 0,C 180,E1 -27847.385,E2 -27847.385} C_VEL
LIN {X 0,Y 80.141,Z 231.318,A -85,B 0,C 180,E1 -27850.709,E2 -27850.709} C_VEL
LIN {X 0,Y 79.699,Z 231.365,A -85,B 0,C 180,E1 -27855.128,E2 -27855.128} C_VEL
LIN {X 0,Y 79.444,Z 231.399,A -85,B 0,C 180,E1 -27862.769,E2 -27862.769} C_VEL
LIN {X 0,Y 79.486,Z 231.39,A -85,B 0,C 180,E1 -27872.153,E2 -27872.153} C_VEL
LIN {X 0,Y 79.517,Z 231.39,A -85,B 0,C 180,E1 -27879.292,E2 -27879.292} C_VEL
LIN {X 0,Y 79.828,Z 231.354,A -85,B 0,C 180,E1 -27885.569,E2 -27885.569} C_VEL
LIN {X 0,Y 79.971,Z 231.328,A -85,B 0,C 180,E1 -27889.873,E2 -27889.873} C_VEL
LIN {X 0,Y 80.647,Z 231.248,A -85,B 0,C 180,E1 -27899.996,E2 -27899.996} C_VEL
LIN {X 0,Y 79.945,Z 231.339,A -85,B 0,C 180,E1 -27910.122,E2 -27910.122} C_VEL
LIN {X 0,Y 79.692,Z 231.363,A -85,B 0,C 180,E1 -27915.337,E2 -27915.337} C_VEL
LIN {X 0,Y 79.497,Z 231.393,A -85,B 0,C 180,E1 -27920.704,E2 -27920.704} C_VEL
LIN {X 0,Y 79.482,Z 231.397,A -85,B 0,C 180,E1 -27927.842,E2 -27927.842} C_VEL
LIN {X 0,Y 79.383,Z 231.401,A -85,B 0,C 180,E1 -27932.081,E2 -27932.081} C_VEL
LIN {X 0,Y 79.37,Z 231.407,A -85,B 0,C 180,E1 -27938.298,E2 -27938.298} C_VEL
LIN {X 0,Y 79.406,Z 231.406,A -85,B 0,C 180,E1 -27945.07,E2 -27945.07} C_VEL
LIN {X 0,Y 79.381,Z 231.409,A -85,B 0,C 180,E1 -27952.819,E2 -27952.819} C_VEL
LIN {X 0,Y 79.373,Z 231.404,A -85,B 0,C 180,E1 -27957.908,E2 -27957.908} C_VEL
LIN {X 0,Y 79.52,Z 231.387,A -85,B 0,C 180,E1 -27963.774,E2 -27963.774} C_VEL
LIN {X 0,Y 79.517,Z 231.393,A -85,B 0,C 180,E1 -27969.295,E2 -27969.295} C_VEL
LIN {X 0,Y 79.836,Z 231.349,A -85,B 0,C 180,E1 -27975.523,E2 -27975.523} C_VEL
LIN {X 0,Y 79.987,Z 231.331,A -85,B 0,C 180,E1 -27979.878,E2 -27979.878} C_VEL
LIN {X 0,Y 80.629,Z 231.246,A -85,B 0,C 180,E1 -27989.999,E2 -27989.999} C_VEL
LIN {X 0,Y 79.823,Z 231.348,A -85,B 0,C 180,E1 -27999.501,E2 -27999.501} C_VEL
LIN {X 0,Y 81.206,Z 238.292,A -85,B 0,C 180,E1 -28001.633,E2 -28001.633} C_VEL
LIN {X 0,Y 82.072,Z 247.736,A -85,B 0,C 180,E1 -28004.885,E2 -28004.885} C_VEL
LIN {X 0,Y 82.675,Z 256.787,A -85,B 0,C 180,E1 -28008.66,E2 -28008.66} C_VEL
LIN {X 0,Y 82.758,Z 258.187,A -85,B 0,C 180,E1 -28009.284,E2 -28009.284} C_VEL
LIN {X 0,Y 82.357,Z 261.403,A -85,B 0,C 180,E1 -28010.776,E2 -28010.776} C_VEL
LIN {X 0,Y 81.17,Z 264.489,A -85,B 0,C 180,E1 -28012.238,E2 -28012.238} C_VEL
LIN {X 0,Y 77.466,Z 270.151,A -85,B 0,C 180,E1 -28015.267,E2 -28015.267} C_VEL
LIN {X 0,Y 72.513,Z 276.666,A -85,B 0,C 180,E1 -28019.969,E2 -28019.969} C_VEL
LIN {X 0,Y 70.872,Z 280.46,A -85,B 0,C 180,E1 -28023.533,E2 -28023.533} C_VEL
LIN {X 0,Y 69.832,Z 287.032,A -85,B 0,C 180,E1 -28030.855,E2 -28030.855} C_VEL
LIN {X 0,Y 69.829,Z 292.859,A -85,B 0,C 180,E1 -28039.148,E2 -28039.148} C_VEL
LIN {X 0,Y 71.054,Z 297.168,A -85,B 0,C 180,E1 -28047.049,E2 -28047.049} C_VEL
LIN {X 0,Y 73.597,Z 300.338,A -85,B 0,C 180,E1 -28054.656,E2 -28054.656} C_VEL
LIN {X 0,Y 75.495,Z 301.63,A -85,B 0,C 180,E1 -28058.577,E2 -28058.577} C_VEL
LIN {X 0,Y 79.944,Z 303.31,A -85,B 0,C 180,E1 -28065.243,E2 -28065.243} C_VEL
LIN {X 0,Y 85.351,Z 303.999,A -85,B 0,C 180,E1 -28071.151,E2 -28071.151} C_VEL
LIN {X 0,Y 91.557,Z 303.696,A -85,B 0,C 180,E1 -28076.267,E2 -28076.267} C_VEL
LIN {X 0,Y 98.398,Z 302.417,A -85,B 0,C 180,E1 -28080.661,E2 -28080.661} C_VEL
LIN {X 0,Y 104.348,Z 300.698,A -85,B 0,C 180,E1 -28083.865,E2 -28083.865} C_VEL
LIN {X 0,Y 105.984,Z 299.921,A -85,B 0,C 180,E1 -28085.921,E2 -28085.921} C_VEL
LIN {X 0,Y 106.877,Z 299.465,A -85,B 0,C 180,E1 -28087.56,E2 -28087.56} C_VEL
LIN {X 0,Y 107.718,Z 298.856,A -85,B 0,C 180,E1 -28091.86,E2 -28091.86} C_VEL
LIN {X 0,Y 107.932,Z 298.627,A -85,B 0,C 180,E1 -28095.101,E2 -28095.101} C_VEL
LIN {X 0,Y 107.907,Z 298.656,A -85,B 0,C 180,E1 -28099.008,E2 -28099.008} C_VEL
LIN {X 0,Y 107.697,Z 299.167,A -85,B 0,C 180,E1 -28103.993,E2 -28103.993} C_VEL
LIN {X 0,Y 107.322,Z 299.809,A -85,B 0,C 180,E1 -28107.287,E2 -28107.287} C_VEL
LIN {X 0,Y 106.597,Z 301.029,A -85,B 0,C 180,E1 -28111.836,E2 -28111.836} C_VEL
LIN {X 0,Y 104.999,Z 302.632,A -85,B 0,C 180,E1 -28116.564,E2 -28116.564} C_VEL
LIN {X 0,Y 100.494,Z 304.639,A -85,B 0,C 180,E1 -28119.712,E2 -28119.712} C_VEL
LIN {X 0,Y 95.482,Z 306.264,A -85,B 0,C 180,E1 -28122.604,E2 -28122.604} C_VEL
LIN {X 0,Y 90.698,Z 307.331,A -85,B 0,C 180,E1 -28125.783,E2 -28125.783} C_VEL
LIN {X 0,Y 82.252,Z 308.216,A -85,B 0,C 180,E1 -28133.266,E2 -28133.266} C_VEL
LIN {X 0,Y 78.646,Z 308.033,A -85,B 0,C 180,E1 -28137.577,E2 -28137.577} C_VEL
LIN {X 0,Y 75.774,Z 307.323,A -85,B 0,C 180,E1 -28142.372,E2 -28142.372} C_VEL
LIN {X 0,Y 73.483,Z 306.19,A -85,B 0,C 180,E1 -28147.509,E2 -28147.509} C_VEL
LIN {X 0,Y 71.315,Z 303.658,A -85,B 0,C 180,E1 -28155.738,E2 -28155.738} C_VEL
LIN {X 0,Y 70.812,Z 300.035,A -85,B 0,C 180,E1 -28164.305,E2 -28164.305} C_VEL
LIN {X 0,Y 70.881,Z 296.754,A -85,B 0,C 180,E1 -28170.001,E2 -28170.001} C_VEL
LIN {X 0,Y 70.961,Z 290.286,A -85,B 0,C 180,E1 -28178.542,E2 -28178.542} C_VEL
LIN {X 0,Y 71.926,Z 283.102,A -85,B 0,C 180,E1 -28185.589,E2 -28185.589} C_VEL
LIN {X 0,Y 73.375,Z 276.01,A -85,B 0,C 180,E1 -28191.051,E2 -28191.051} C_VEL
LIN {X 0,Y 73.742,Z 270.377,A -85,B 0,C 180,E1 -28194.644,E2 -28194.644} C_VEL
LIN {X 0,Y 74.001,Z 261.467,A -85,B 0,C 180,E1 -28199.37,E2 -28199.37} C_VEL
LIN {X 0,Y 74.299,Z 251.435,A -85,B 0,C 180,E1 -28203.612,E2 -28203.612} C_VEL
LIN {X 0,Y 74.433,Z 239.539,A -85,B 0,C 180,E1 -28207.301,E2 -28207.301} C_VEL
LIN {X 0,Y 74.077,Z 236.209,A -85,B 0,C 180,E1 -28208.244,E2 -28208.244} C_VEL
LIN {X 0,Y 73.127,Z 232.25,A -85,B 0,C 180,E1 -28209.477,E2 -28209.477} C_VEL
LIN {X 0,Y 72.454,Z 232.265,A -85,B 0,C 180,E1 -28217.229,E2 -28217.229} C_VEL
LIN {X 0,Y 72.332,Z 232.279,A -85,B 0,C 180,E1 -28224.335,E2 -28224.335} C_VEL
LIN {X 0,Y 72.379,Z 232.279,A -85,B 0,C 180,E1 -28230.95,E2 -28230.95} C_VEL
LIN {X 0,Y 72.398,Z 232.279,A -85,B 0,C 180,E1 -28237.146,E2 -28237.146} C_VEL
LIN {X 0,Y 72.725,Z 232.238,A -85,B 0,C 180,E1 -28245.105,E2 -28245.105} C_VEL
LIN {X 0,Y 72.862,Z 232.215,A -85,B 0,C 180,E1 -28248.872,E2 -28248.872} C_VEL
LIN {X 0,Y 73.572,Z 232.128,A -85,B 0,C 180,E1 -28259.995,E2 -28259.995} C_VEL
LIN {X 0,Y 72.832,Z 232.225,A -85,B 0,C 180,E1 -28271.123,E2 -28271.123} C_VEL
LIN {X 0,Y 72.513,Z 232.261,A -85,B 0,C 180,E1 -28276.898,E2 -28276.898} C_VEL
LIN {X 0,Y 72.385,Z 232.273,A -85,B 0,C 180,E1 -28282.848,E2 -28282.848} C_VEL
LIN {X 0,Y 72.375,Z 232.281,A -85,B 0,C 180,E1 -28289.077,E2 -28289.077} C_VEL
LIN {X 0,Y 72.298,Z 232.292,A -85,B 0,C 180,E1 -28295.673,E2 -28295.673} C_VEL
LIN {X 0,Y 72.258,Z 232.296,A -85,B 0,C 180,E1 -28302.902,E2 -28302.902} C_VEL
LIN {X 0,Y 72.291,Z 232.291,A -85,B 0,C 180,E1 -28311.046,E2 -28311.046} C_VEL
LIN {X 0,Y 72.289,Z 232.291,A -85,B 0,C 180,E1 -28314.314,E2 -28314.314} C_VEL
LIN {X 0,Y 72.37,Z 232.283,A -85,B 0,C 180,E1 -28320.949,E2 -28320.949} C_VEL
LIN {X 0,Y 72.394,Z 232.276,A -85,B 0,C 180,E1 -28327.149,E2 -28327.149} C_VEL
LIN {X 0,Y 72.752,Z 232.23,A -85,B 0,C 180,E1 -28335.002,E2 -28335.002} C_VEL
LIN {X 0,Y 72.874,Z 232.219,A -85,B 0,C 180,E1 -28338.878,E2 -28338.878} C_VEL
LIN {X 0,Y 73.549,Z 232.128,A -85,B 0,C 180,E1 -28349.999,E2 -28349.999} C_VEL
LIN {X 0,Y 72.83,Z 232.271,A -85,B 0,C 180,E1 -28357.798,E2 -28357.798} C_VEL
LIN {X 0,Y 74.42,Z 239.111,A -85,B 0,C 180,E1 -28360.198,E2 -28360.198} C_VEL
LIN {X 0,Y 75.119,Z 247.976,A -85,B 0,C 180,E1 -28363.525,E2 -28363.525} C_VEL
LIN {X 0,Y 75.675,Z 256.874,A -85,B 0,C 180,E1 -28367.566,E2 -28367.566} C_VEL
LIN {X 0,Y 75.804,Z 259.634,A -85,B 0,C 180,E1 -28368.934,E2 -28368.934} C_VEL
LIN {X 0,Y 73.71,Z 268.354,A -85,B 0,C 180,E1 -28373.904,E2 -28373.904} C_VEL
LIN {X 0,Y 71.903,Z 275.669,A -85,B 0,C 180,E1 -28379.255,E2 -28379.255} C_VEL
LIN {X 0,Y 70.872,Z 280.46,A -85,B 0,C 180,E1 -28383.533,E2 -28383.533} C_VEL
LIN {X 0,Y 69.593,Z 284.056,A -85,B 0,C 180,E1 -28387.279,E2 -28387.279} C_VEL
LIN {X 0,Y 66.187,Z 288.988,A -85,B 0,C 180,E1 -28393.929,E2 -28393.929} C_VEL
LIN {X 0,Y 63.635,Z 293.299,A -85,B 0,C 180,E1 -28401.573,E2 -28401.573} C_VEL
LIN {X 0,Y 63.731,Z 295.651,A -85,B 0,C 180,E1 -28406.477,E2 -28406.477} C_VEL
LIN {X 0,Y 66.23,Z 299.315,A -85,B 0,C 180,E1 -28414.89,E2 -28414.89} C_VEL
LIN {X 0,Y 69.944,Z 301.915,A -85,B 0,C 180,E1 -28422.461,E2 -28422.461} C_VEL
LIN {X 0,Y 74.888,Z 303.593,A -85,B 0,C 180,E1 -28429.187,E2 -28429.187} C_VEL
LIN {X 0,Y 80.713,Z 304.34,A -85,B 0,C 180,E1 -28435.009,E2 -28435.009} C_VEL
LIN {X 0,Y 87.321,Z 304.163,A -85,B 0,C 180,E1 -28440.004,E2 -28440.004} C_VEL
LIN {X 0,Y 94.602,Z 303.039,A -85,B 0,C 180,E1 -28444.264,E2 -28444.264} C_VEL
LIN {X 0,Y 99.079,Z 301.876,A -85,B 0,C 180,E1 -28446.758,E2 -28446.758} C_VEL
LIN {X 0,Y 100.029,Z 301.601,A -85,B 0,C 180,E1 -28448.081,E2 -28448.081} C_VEL
LIN {X 0,Y 101.011,Z 301.122,A -85,B 0,C 180,E1 -28452.051,E2 -28452.051} C_VEL
LIN {X 0,Y 101.214,Z 301.028,A -85,B 0,C 180,E1 -28456.129,E2 -28456.129} C_VEL
LIN {X 0,Y 101.141,Z 301.213,A -85,B 0,C 180,E1 -28460.334,E2 -28460.334} C_VEL
LIN {X 0,Y 100.831,Z 301.763,A -85,B 0,C 180,E1 -28465.028,E2 -28465.028} C_VEL
LIN {X 0,Y 100.144,Z 302.607,A -85,B 0,C 180,E1 -28469.427,E2 -28469.427} C_VEL
LIN {X 0,Y 99.499,Z 303.299,A -85,B 0,C 180,E1 -28472.049,E2 -28472.049} C_VEL
LIN {X 0,Y 98.56,Z 304.052,A -85,B 0,C 180,E1 -28474.786,E2 -28474.786} C_VEL
LIN {X 0,Y 96.053,Z 304.877,A -85,B 0,C 180,E1 -28476.406,E2 -28476.406} C_VEL
LIN {X 0,Y 90.828,Z 306.292,A -85,B 0,C 180,E1 -28479.308,E2 -28479.308} C_VEL
LIN {X 0,Y 85.747,Z 307.29,A -85,B 0,C 180,E1 -28482.469,E2 -28482.469} C_VEL
LIN {X 0,Y 81.042,Z 307.748,A -85,B 0,C 180,E1 -28486.072,E2 -28486.072} C_VEL
LIN {X 0,Y 72.763,Z 307.411,A -85,B 0,C 180,E1 -28494.584,E2 -28494.584} C_VEL
LIN {X 0,Y 69.576,Z 306.651,A -85,B 0,C 180,E1 -28499.666,E2 -28499.666} C_VEL
LIN {X 0,Y 67.006,Z 305.348,A -85,B 0,C 180,E1 -28505.195,E2 -28505.195} C_VEL
LIN {X 0,Y 64.518,Z 302.616,A -85,B 0,C 180,E1 -28514.198,E2 -28514.198} C_VEL
LIN {X 0,Y 63.859,Z 298.687,A -85,B 0,C 180,E1 -28523.683,E2 -28523.683} C_VEL
LIN {X 0,Y 63.874,Z 295.239,A -85,B 0,C 180,E1 -28530.001,E2 -28530.001} C_VEL
LIN {X 0,Y 63.949,Z 289.158,A -85,B 0,C 180,E1 -28538.433,E2 -28538.433} C_VEL
LIN {X 0,Y 64.879,Z 282.417,A -85,B 0,C 180,E1 -28545.714,E2 -28545.714} C_VEL
LIN {X 0,Y 66.372,Z 275.292,A -85,B 0,C 180,E1 -28551.754,E2 -28551.754} C_VEL
LIN {X 0,Y 66.693,Z 269.522,A -85,B 0,C 180,E1 -28555.766,E2 -28555.766} C_VEL
LIN {X 0,Y 67.071,Z 260.97,A -85,B 0,C 180,E1 -28560.72,E2 -28560.72} C_VEL
LIN {X 0,Y 67.463,Z 250.561,A -85,B 0,C 180,E1 -28565.521,E2 -28565.521} C_VEL
LIN {X 0,Y 67.712,Z 239.424,A -85,B 0,C 180,E1 -28569.263,E2 -28569.263} C_VEL
LIN {X 0,Y 66.399,Z 234.878,A -85,B 0,C 180,E1 -28570.981,E2 -28570.981} C_VEL
LIN {X 0,Y 65.903,Z 233.089,A -85,B 0,C 180,E1 -28571.705,E2 -28571.705} C_VEL
LIN {X 0,Y 65.334,Z 233.159,A -85,B 0,C 180,E1 -28579.796,E2 -28579.796} C_VEL
LIN {X 0,Y 65.263,Z 233.168,A -85,B 0,C 180,E1 -28589.488,E2 -28589.488} C_VEL
LIN {X 0,Y 65.242,Z 233.164,A -85,B 0,C 180,E1 -28594.47,E2 -28594.47} C_VEL
LIN {X 0,Y 65.629,Z 233.122,A -85,B 0,C 180,E1 -28604.538,E2 -28604.538} C_VEL
LIN {X 0,Y 65.759,Z 233.103,A -85,B 0,C 180,E1 -28607.652,E2 -28607.652} C_VEL
LIN {X 0,Y 66.494,Z 233.009,A -85,B 0,C 180,E1 -28619.995,E2 -28619.995} C_VEL
LIN {X 0,Y 65.724,Z 233.109,A -85,B 0,C 180,E1 -28632.343,E2 -28632.343} C_VEL
LIN {X 0,Y 65.346,Z 233.158,A -85,B 0,C 180,E1 -28638.818,E2 -28638.818} C_VEL
LIN {X 0,Y 65.241,Z 233.167,A -85,B 0,C 180,E1 -28645.518,E2 -28645.518} C_VEL
LIN {X 0,Y 65.196,Z 233.169,A -85,B 0,C 180,E1 -28652.608,E2 -28652.608} C_VEL
LIN {X 0,Y 65.19,Z 233.17,A -85,B 0,C 180,E1 -28661.003,E2 -28661.003} C_VEL
LIN {X 0,Y 65.204,Z 233.169,A -85,B 0,C 180,E1 -28669.704,E2 -28669.704} C_VEL
LIN {X 0,Y 65.249,Z 233.168,A -85,B 0,C 180,E1 -28679.495,E2 -28679.495} C_VEL
LIN {X 0,Y 65.235,Z 233.164,A -85,B 0,C 180,E1 -28684.472,E2 -28684.472} C_VEL
LIN {X 0,Y 65.646,Z 233.113,A -85,B 0,C 180,E1 -28694.458,E2 -28694.458} C_VEL
LIN {X 0,Y 65.775,Z 233.105,A -85,B 0,C 180,E1 -28697.66,E2 -28697.66} C_VEL
LIN {X 0,Y 65.927,Z 233.081,A -85,B 0,C 180,E1 -28703.879,E2 -28703.879} C_VEL
LIN {X 0,Y 66.44,Z 233.013,A -85,B 0,C 180,E1 -28709.999,E2 -28709.999} C_VEL
LIN {X 0,Y 65.9,Z 233.166,A -85,B 0,C 180,E1 -28715.737,E2 -28715.737} C_VEL
LIN {X 0,Y 67.491,Z 239.231,A -85,B 0,C 180,E1 -28718.231,E2 -28718.231} C_VEL
LIN {X 0,Y 68.223,Z 247.968,A -85,B 0,C 180,E1 -28721.889,E2 -28721.889} C_VEL
LIN {X 0,Y 68.645,Z 256.925,A -85,B 0,C 180,E1 -28726.352,E2 -28726.352} C_VEL
LIN {X 0,Y 68.765,Z 259.693,A -85,B 0,C 180,E1 -28727.854,E2 -28727.854} C_VEL
LIN {X 0,Y 66.83,Z 267.565,A -85,B 0,C 180,E1 -28732.656,E2 -28732.656} C_VEL
LIN {X 0,Y 64.853,Z 275.191,A -85,B 0,C 180,E1 -28738.666,E2 -28738.666} C_VEL
LIN {X 0,Y 63.549,Z 281.252,A -85,B 0,C 180,E1 -28744.698,E2 -28744.698} C_VEL
LIN {X 0,Y 62.691,Z 287.305,A -85,B 0,C 180,E1 -28752.269,E2 -28752.269} C_VEL
LIN {X 0,Y 62.825,Z 292.15,A -85,B 0,C 180,E1 -28759.821,E2 -28759.821} C_VEL
LIN {X 0,Y 63.731,Z 295.651,A -85,B 0,C 180,E1 -28766.477,E2 -28766.477} C_VEL
LIN {X 0,Y 64.297,Z 297.826,A -85,B 0,C 180,E1 -28771.385,E2 -28771.385} C_VEL
LIN {X 0,Y 64.623,Z 300.587,A -85,B 0,C 180,E1 -28779.857,E2 -28779.857} C_VEL
LIN {X 0,Y 66.452,Z 302.7,A -85,B 0,C 180,E1 -28788.209,E2 -28788.209} C_VEL
LIN {X 0,Y 69.185,Z 303.56,A -85,B 0,C 180,E1 -28792.557,E2 -28792.557} C_VEL
LIN {X 0,Y 77.395,Z 304.726,A -85,B 0,C 180,E1 -28800.004,E2 -28800.004} C_VEL
LIN {X 0,Y 84.667,Z 304.518,A -85,B 0,C 180,E1 -28804.765,E2 -28804.765} C_VEL
LIN {X 0,Y 92.471,Z 303.357,A -85,B 0,C 180,E1 -28808.879,E2 -28808.879} C_VEL
LIN {X 0,Y 94.189,Z 302.939,A -85,B 0,C 180,E1 -28812.939,E2 -28812.939} C_VEL
LIN {X 0,Y 94.325,Z 303.027,A -85,B 0,C 180,E1 -28817.343,E2 -28817.343} C_VEL
LIN {X 0,Y 94.158,Z 303.348,A -85,B 0,C 180,E1 -28821.917,E2 -28821.917} C_VEL
LIN {X 0,Y 93.592,Z 303.952,A -85,B 0,C 180,E1 -28826.783,E2 -28826.783} C_VEL
LIN {X 0,Y 92.303,Z 304.963,A -85,B 0,C 180,E1 -28832.211,E2 -28832.211} C_VEL
LIN {X 0,Y 91.943,Z 305.128,A -85,B 0,C 180,E1 -28832.774,E2 -28832.774} C_VEL
LIN {X 0,Y 86.505,Z 306.304,A -85,B 0,C 180,E1 -28835.666,E2 -28835.666} C_VEL
LIN {X 0,Y 81.12,Z 307.091,A -85,B 0,C 180,E1 -28838.765,E2 -28838.765} C_VEL
LIN {X 0,Y 76.087,Z 307.483,A -85,B 0,C 180,E1 -28842.36,E2 -28842.36} C_VEL
LIN {X 0,Y 71.411,Z 307.341,A -85,B 0,C 180,E1 -28846.457,E2 -28846.457} C_VEL
LIN {X 0,Y 67.117,Z 306.758,A -85,B 0,C 180,E1 -28851.078,E2 -28851.078} C_VEL
LIN {X 0,Y 63.566,Z 305.805,A -85,B 0,C 180,E1 -28856.441,E2 -28856.441} C_VEL
LIN {X 0,Y 60.665,Z 304.438,A -85,B 0,C 180,E1 -28862.395,E2 -28862.395} C_VEL
LIN {X 0,Y 57.824,Z 301.402,A -85,B 0,C 180,E1 -28872.312,E2 -28872.312} C_VEL
LIN {X 0,Y 56.97,Z 297.201,A -85,B 0,C 180,E1 -28882.915,E2 -28882.915} C_VEL
LIN {X 0,Y 56.89,Z 293.53,A -85,B 0,C 180,E1 -28890.001,E2 -28890.001} C_VEL
LIN {X 0,Y 56.99,Z 287.421,A -85,B 0,C 180,E1 -28899.046,E2 -28899.046} C_VEL
LIN {X 0,Y 57.824,Z 281.644,A -85,B 0,C 180,E1 -28905.872,E2 -28905.872} C_VEL
LIN {X 0,Y 59.376,Z 274.434,A -85,B 0,C 180,E1 -28912.625,E2 -28912.625} C_VEL
LIN {X 0,Y 59.796,Z 265.907,A -85,B 0,C 180,E1 -28919.003,E2 -28919.003} C_VEL
LIN {X 0,Y 60.386,Z 255.872,A -85,B 0,C 180,E1 -28924.802,E2 -28924.802} C_VEL
LIN {X 0,Y 60.779,Z 247.256,A -85,B 0,C 180,E1 -28928.727,E2 -28928.727} C_VEL
LIN {X 0,Y 60.926,Z 240.09,A -85,B 0,C 180,E1 -28931.419,E2 -28931.419} C_VEL
LIN {X 0,Y 59.547,Z 236.645,A -85,B 0,C 180,E1 -28933.083,E2 -28933.083} C_VEL
LIN {X 0,Y 58.503,Z 234.005,A -85,B 0,C 180,E1 -28934.66,E2 -28934.66} C_VEL
LIN {X 0,Y 58.172,Z 234.05,A -85,B 0,C 180,E1 -28947.749,E2 -28947.749} C_VEL
LIN {X 0,Y 58.157,Z 234.049,A -85,B 0,C 180,E1 -28951.087,E2 -28951.087} C_VEL
LIN {X 0,Y 58.52,Z 234.005,A -85,B 0,C 180,E1 -28963.901,E2 -28963.901} C_VEL
LIN {X 0,Y 58.803,Z 233.972,A -85,B 0,C 180,E1 -28973.13,E2 -28973.13} C_VEL
LIN {X 0,Y 59.383,Z 233.895,A -85,B 0,C 180,E1 -28979.994,E2 -28979.994} C_VEL
LIN {X 0,Y 58.786,Z 233.966,A -85,B 0,C 180,E1 -28986.86,E2 -28986.86} C_VEL
LIN {X 0,Y 58.465,Z 234.007,A -85,B 0,C 180,E1 -28995.91,E2 -28995.91} C_VEL
LIN {X 0,Y 58.151,Z 234.053,A -85,B 0,C 180,E1 -29008.903,E2 -29008.903} C_VEL
LIN {X 0,Y 58.157,Z 234.044,A -85,B 0,C 180,E1 -29012.228,E2 -29012.228} C_VEL
LIN {X 0,Y 58.035,Z 234.067,A -85,B 0,C 180,E1 -29017.257,E2 -29017.257} C_VEL
LIN {X 0,Y 58.015,Z 234.066,A -85,B 0,C 180,E1 -29026.613,E2 -29026.613} C_VEL
LIN {X 0,Y 58.03,Z 234.069,A -85,B 0,C 180,E1 -29032.73,E2 -29032.73} C_VEL
LIN {X 0,Y 58.153,Z 234.046,A -85,B 0,C 180,E1 -29037.765,E2 -29037.765} C_VEL
